Fanuc TP program (LS listing): test_parallel_centered.ls

/PROG  test_parallel_centered
/ATTR
COMMENT	= "19-02-13 13:08:30";
PROG_SIZE	= 0;
DEFAULT_GROUP	= 1, 1, *, *, *;
/APPL
    ARC Welding Equipment: 1, *, *, *, *;
/MN
   1:  CALL HOME_ALL;
   1:  UFRAME_NUM = 1;
   1:  UTOOL_NUM = 3;
   1:  COL GUARD ADJUST 150;
   1:  PR[91] = PR[90];
   1:  ! Sicherheitspunkt;
   1:  PR[92] = PR[90];
   1:  PR[92] = PR[GP1:92,3] + 50;
   1:J PR[92];
   1:  PR[GP1:91,1] = PR[GP1:90,1] + -24.070;
   1:  PR[GP1:91,2] = PR[GP1:90,2] + -16.563;
   1:  PR[GP1:91,3] = PR[GP1:90,3] + 1.100;
   1:L PR[91] 10mm/sec CNT100;
   1:  PR[GP1:91,1] = PR[GP1:90,1] + -23.760;
   1:  PR[GP1:91,2] = PR[GP1:90,2] + -16.616;
   1:L PR[91] 10mm/sec CNT100;
   1:  PR[GP1:91,1] = PR[GP1:90,1] + -18.882;
   1:  PR[GP1:91,2] = PR[GP1:90,2] + -17.045;
   1:L PR[91] 10mm/sec CNT100;
   1:  PR[GP1:91,1] = PR[GP1:90,1] + -18.568;
   1:  PR[GP1:91,2] = PR[GP1:90,2] + -17.047;
   1:L PR[91] 10mm/sec CNT100;
   1:  PR[GP1:91,1] = PR[GP1:90,1] + -18.257;
   1:  PR[GP1:91,2] = PR[GP1:90,2] + -16.997;
   1:L PR[91] 10mm/sec CNT100;
   1:  PR[GP1:91,1] = PR[GP1:90,1] + -13.503;
   1:  PR[GP1:91,2] = PR[GP1:90,2] + -15.824;
   1:L PR[91] 10mm/sec CNT100;
   1:  PR[GP1:91,1] = PR[GP1:90,1] + -13.205;
   1:  PR[GP1:91,2] = PR[GP1:90,2] + -15.724;
   1:L PR[91] 10mm/sec CNT100;
   1:  PR[GP1:91,1] = PR[GP1:90,1] + -12.928;
   1:  PR[GP1:91,2] = PR[GP1:90,2] + -15.576;
   1:L PR[91] 10mm/sec CNT100;
   1:  PR[GP1:91,1] = PR[GP1:90,1] + -8.809;
   1:  PR[GP1:91,2] = PR[GP1:90,2] + -12.928;
   1:L PR[91] 10mm/sec CNT100;
   1:  PR[GP1:91,1] = PR[GP1:90,1] + -8.559;
   1:  PR[GP1:91,2] = PR[GP1:90,2] + -12.737;
   1:L PR[91] 10mm/sec CNT100;
   1:  PR[GP1:91,1] = PR[GP1:90,1] + -8.344;
   1:  PR[GP1:91,2] = PR[GP1:90,2] + -12.508;
   1:L PR[91] 10mm/sec CNT100;
   1:  PR[GP1:91,1] = PR[GP1:90,1] + -5.304;
   1:  PR[GP1:91,2] = PR[GP1:90,2] + -8.669;
   1:L PR[91] 10mm/sec CNT100;
   1:  PR[GP1:91,1] = PR[GP1:90,1] + -5.129;
   1:  PR[GP1:91,2] = PR[GP1:90,2] + -8.408;
   1:L PR[91] 10mm/sec CNT100;
   1:  PR[GP1:91,1] = PR[GP1:90,1] + -5.000;
   1:  PR[GP1:91,2] = PR[GP1:90,2] + -8.121;
   1:L PR[91] 10mm/sec CNT100;
   1:  PR[GP1:91,1] = PR[GP1:90,1] + -3.366;
   1:  PR[GP1:91,2] = PR[GP1:90,2] + -3.509;
   1:L PR[91] 10mm/sec CNT100;
   1:  PR[GP1:91,1] = PR[GP1:90,1] + -3.259;
   1:  PR[GP1:91,2] = PR[GP1:90,2] + -3.105;
   1:L PR[91] 10mm/sec CNT100;
   1:  PR[GP1:91,1] = PR[GP1:90,1] + -2.720;
   1:  PR[GP1:91,2] = PR[GP1:90,2] + -1.858;
   1:L PR[91] 10mm/sec CNT100;
   1:  PR[GP1:91,1] = PR[GP1:90,1] + -1.598;
   1:  PR[GP1:91,2] = PR[GP1:90,2] + -0.918;
   1:L PR[91] 10mm/sec CNT100;
   1:  PR[GP1:91,1] = PR[GP1:90,1] + -0.249;
   1:  PR[GP1:91,2] = PR[GP1:90,2] + -0.599;
   1:L PR[91] 10mm/sec CNT100;
   1:  PR[GP1:91,1] = PR[GP1:90,1] + 0.522;
   1:L PR[91] 10mm/sec CNT100;
   1:  PR[GP1:91,1] = PR[GP1:90,1] + 1.871;
   1:  PR[GP1:91,2] = PR[GP1:90,2] + -0.918;
   1:L PR[91] 10mm/sec CNT100;
   1:  PR[GP1:91,1] = PR[GP1:90,1] + 2.993;
   1:  PR[GP1:91,2] = PR[GP1:90,2] + -1.858;
   1:L PR[91] 10mm/sec CNT100;
   1:  PR[GP1:91,1] = PR[GP1:90,1] + 3.521;
   1:  PR[GP1:91,2] = PR[GP1:90,2] + -3.080;
   1:L PR[91] 10mm/sec CNT100;
   1:  PR[GP1:91,1] = PR[GP1:90,1] + 5.193;
   1:  PR[GP1:91,2] = PR[GP1:90,2] + -7.798;
   1:L PR[91] 10mm/sec CNT100;
   1:  PR[GP1:91,1] = PR[GP1:90,1] + 5.253;
   1:  PR[GP1:91,2] = PR[GP1:90,2] + -8.055;
   1:L PR[91] 10mm/sec CNT100;
   1:  PR[GP1:91,1] = PR[GP1:90,1] + 5.317;
   1:  PR[GP1:91,2] = PR[GP1:90,2] + -8.236;
   1:L PR[91] 10mm/sec CNT100;
   1:  PR[GP1:91,1] = PR[GP1:90,1] + 5.385;
   1:  PR[GP1:91,2] = PR[GP1:90,2] + -8.375;
   1:L PR[91] 10mm/sec CNT100;
   1:  PR[GP1:91,1] = PR[GP1:90,1] + 8.437;
   1:  PR[GP1:91,2] = PR[GP1:90,2] + -12.228;
   1:L PR[91] 10mm/sec CNT100;
   1:  PR[GP1:91,1] = PR[GP1:90,1] + 8.577;
   1:  PR[GP1:91,2] = PR[GP1:90,2] + -12.452;
   1:L PR[91] 10mm/sec CNT100;
   1:  PR[GP1:91,1] = PR[GP1:90,1] + 8.696;
   1:  PR[GP1:91,2] = PR[GP1:90,2] + -12.602;
   1:L PR[91] 10mm/sec CNT100;
   1:  PR[GP1:91,1] = PR[GP1:90,1] + 8.805;
   1:  PR[GP1:91,2] = PR[GP1:90,2] + -12.712;
   1:L PR[91] 10mm/sec CNT100;
   1:  PR[GP1:91,1] = PR[GP1:90,1] + 12.939;
   1:  PR[GP1:91,2] = PR[GP1:90,2] + -15.370;
   1:L PR[91] 10mm/sec CNT100;
   1:  PR[GP1:91,1] = PR[GP1:90,1] + 13.144;
   1:  PR[GP1:91,2] = PR[GP1:90,2] + -15.536;
   1:L PR[91] 10mm/sec CNT100;
   1:  PR[GP1:91,1] = PR[GP1:90,1] + 13.306;
   1:  PR[GP1:91,2] = PR[GP1:90,2] + -15.640;
   1:L PR[91] 10mm/sec CNT100;
   1:  PR[GP1:91,1] = PR[GP1:90,1] + 13.444;
   1:  PR[GP1:91,2] = PR[GP1:90,2] + -15.709;
   1:L PR[91] 10mm/sec CNT100;
   1:  PR[GP1:91,1] = PR[GP1:90,1] + 18.216;
   1:  PR[GP1:91,2] = PR[GP1:90,2] + -16.885;
   1:L PR[91] 10mm/sec CNT100;
   1:  PR[GP1:91,1] = PR[GP1:90,1] + 18.464;
   1:  PR[GP1:91,2] = PR[GP1:90,2] + -16.976;
   1:L PR[91] 10mm/sec CNT100;
   1:  PR[GP1:91,1] = PR[GP1:90,1] + 18.650;
   1:  PR[GP1:91,2] = PR[GP1:90,2] + -17.022;
   1:L PR[91] 10mm/sec CNT100;
   1:  PR[GP1:91,1] = PR[GP1:90,1] + 18.803;
   1:  PR[GP1:91,2] = PR[GP1:90,2] + -17.043;
   1:L PR[91] 10mm/sec CNT100;
   1:  PR[GP1:91,1] = PR[GP1:90,1] + 23.699;
   1:  PR[GP1:91,2] = PR[GP1:90,2] + -16.613;
   1:L PR[91] 10mm/sec CNT100;
   1:  PR[GP1:91,1] = PR[GP1:90,1] + 23.963;
   1:  PR[GP1:91,2] = PR[GP1:90,2] + -16.618;
   1:L PR[91] 10mm/sec CNT100;
   1:  PR[GP1:91,1] = PR[GP1:90,1] + 24.154;
   1:  PR[GP1:91,2] = PR[GP1:90,2] + -16.602;
   1:L PR[91] 10mm/sec CNT100;
   1:  PR[GP1:91,1] = PR[GP1:90,1] + 24.306;
   1:  PR[GP1:91,2] = PR[GP1:90,2] + -16.571;
   1:L PR[91] 10mm/sec CNT100;
   1:  PR[GP1:91,1] = PR[GP1:90,1] + 28.799;
   1:  PR[GP1:91,2] = PR[GP1:90,2] + -14.580;
   1:L PR[91] 10mm/sec CNT100;
   1:  PR[GP1:91,1] = PR[GP1:90,1] + 29.051;
   1:  PR[GP1:91,2] = PR[GP1:90,2] + -14.500;
   1:L PR[91] 10mm/sec CNT100;
   1:  PR[GP1:91,1] = PR[GP1:90,1] + 29.226;
   1:  PR[GP1:91,2] = PR[GP1:90,2] + -14.422;
   1:L PR[91] 10mm/sec CNT100;
   1:  PR[GP1:91,1] = PR[GP1:90,1] + 29.360;
   1:  PR[GP1:91,2] = PR[GP1:90,2] + -14.344;
   1:L PR[91] 10mm/sec CNT100;
   1:  PR[GP1:91,1] = PR[GP1:90,1] + 32.968;
   1:  PR[GP1:91,2] = PR[GP1:90,2] + -11.006;
   1:L PR[91] 10mm/sec CNT100;
   1:  PR[GP1:91,1] = PR[GP1:90,1] + 33.180;
   1:  PR[GP1:91,2] = PR[GP1:90,2] + -10.849;
   1:L PR[91] 10mm/sec CNT100;
   1:  PR[GP1:91,1] = PR[GP1:90,1] + 33.321;
   1:  PR[GP1:91,2] = PR[GP1:90,2] + -10.719;
   1:L PR[91] 10mm/sec CNT100;
   1:  PR[GP1:91,1] = PR[GP1:90,1] + 33.422;
   1:  PR[GP1:91,2] = PR[GP1:90,2] + -10.601;
   1:L PR[91] 10mm/sec CNT100;
   1:  PR[GP1:91,1] = PR[GP1:90,1] + 35.756;
   1:  PR[GP1:91,2] = PR[GP1:90,2] + -6.274;
   1:L PR[91] 10mm/sec CNT100;
   1:  PR[GP1:91,1] = PR[GP1:90,1] + 35.906;
   1:  PR[GP1:91,2] = PR[GP1:90,2] + -6.057;
   1:L PR[91] 10mm/sec CNT100;
   1:  PR[GP1:91,1] = PR[GP1:90,1] + 35.997;
   1:  PR[GP1:91,2] = PR[GP1:90,2] + -5.888;
   1:L PR[91] 10mm/sec CNT100;
   1:  PR[GP1:91,1] = PR[GP1:90,1] + 36.055;
   1:  PR[GP1:91,2] = PR[GP1:90,2] + -5.744;
   1:L PR[91] 10mm/sec CNT100;
   1:  PR[GP1:91,1] = PR[GP1:90,1] + 36.862;
   1:  PR[GP1:91,2] = PR[GP1:90,2] + -0.893;
   1:L PR[91] 10mm/sec CNT100;
   1:  PR[GP1:91,1] = PR[GP1:90,1] + 36.933;
   1:  PR[GP1:91,2] = PR[GP1:90,2] + -0.639;
   1:L PR[91] 10mm/sec CNT100;
   1:  PR[GP1:91,1] = PR[GP1:90,1] + 36.965;
   1:  PR[GP1:91,2] = PR[GP1:90,2] + -0.450;
   1:L PR[91] 10mm/sec CNT100;
   1:  PR[GP1:91,1] = PR[GP1:90,1] + 36.973;
   1:  PR[GP1:91,2] = PR[GP1:90,2] + -0.295;
   1:L PR[91] 10mm/sec CNT100;
   1:  PR[GP1:91,1] = PR[GP1:90,1] + 36.169;
   1:  PR[GP1:91,2] = PR[GP1:90,2] + 4.541;
   1:L PR[91] 10mm/sec CNT100;
   1:  PR[GP1:91,1] = PR[GP1:90,1] + 36.125;
   1:  PR[GP1:91,2] = PR[GP1:90,2] + 4.981;
   1:L PR[91] 10mm/sec CNT100;
   1:  PR[GP1:91,1] = PR[GP1:90,1] + 36.065;
   1:  PR[GP1:91,2] = PR[GP1:90,2] + 5.203;
   1:L PR[91] 10mm/sec CNT100;
   1:  PR[GP1:91,1] = PR[GP1:90,1] + 36.036;
   1:  PR[GP1:91,2] = PR[GP1:90,2] + 5.281;
   1:L PR[91] 10mm/sec CNT100;
   1:  PR[GP1:91,1] = PR[GP1:90,1] + 33.501;
   1:  PR[GP1:91,2] = PR[GP1:90,2] + 9.982;
   1:L PR[91] 10mm/sec CNT100;
   1:  PR[GP1:91,1] = PR[GP1:90,1] + 33.453;
   1:  PR[GP1:91,2] = PR[GP1:90,2] + 10.048;
   1:L PR[91] 10mm/sec CNT100;
   1:  PR[GP1:91,1] = PR[GP1:90,1] + 33.285;
   1:  PR[GP1:91,2] = PR[GP1:90,2] + 10.237;
   1:L PR[91] 10mm/sec CNT100;
   1:  PR[GP1:91,1] = PR[GP1:90,1] + 29.691;
   1:  PR[GP1:91,2] = PR[GP1:90,2] + 13.563;
   1:L PR[91] 10mm/sec CNT100;
   1:  PR[GP1:91,1] = PR[GP1:90,1] + 29.406;
   1:  PR[GP1:91,2] = PR[GP1:90,2] + 13.794;
   1:L PR[91] 10mm/sec CNT100;
   1:  PR[GP1:91,1] = PR[GP1:90,1] + 24.940;
   1:  PR[GP1:91,2] = PR[GP1:90,2] + 15.773;
   1:L PR[91] 10mm/sec CNT100;
   1:  PR[GP1:91,1] = PR[GP1:90,1] + 24.548;
   1:  PR[GP1:91,2] = PR[GP1:90,2] + 15.978;
   1:L PR[91] 10mm/sec CNT100;
   1:  PR[GP1:91,1] = PR[GP1:90,1] + 24.331;
   1:  PR[GP1:91,2] = PR[GP1:90,2] + 16.049;
   1:L PR[91] 10mm/sec CNT100;
   1:  PR[GP1:91,1] = PR[GP1:90,1] + 24.248;
   1:  PR[GP1:91,2] = PR[GP1:90,2] + 16.068;
   1:L PR[91] 10mm/sec CNT100;
   1:  PR[GP1:91,1] = PR[GP1:90,1] + 18.930;
   1:  PR[GP1:91,2] = PR[GP1:90,2] + 16.535;
   1:L PR[91] 10mm/sec CNT100;
   1:  PR[GP1:91,1] = PR[GP1:90,1] + 18.851;
   1:  PR[GP1:91,2] = PR[GP1:90,2] + 16.531;
   1:L PR[91] 10mm/sec CNT100;
   1:  PR[GP1:91,1] = PR[GP1:90,1] + 18.598;
   1:  PR[GP1:91,2] = PR[GP1:90,2] + 16.495;
   1:L PR[91] 10mm/sec CNT100;
   1:  PR[GP1:91,1] = PR[GP1:90,1] + 13.844;
   1:  PR[GP1:91,2] = PR[GP1:90,2] + 15.322;
   1:L PR[91] 10mm/sec CNT100;
   1:  PR[GP1:91,1] = PR[GP1:90,1] + 13.499;
   1:  PR[GP1:91,2] = PR[GP1:90,2] + 15.212;
   1:L PR[91] 10mm/sec CNT100;
   1:  PR[GP1:91,1] = PR[GP1:90,1] + 9.386;
   1:  PR[GP1:91,2] = PR[GP1:90,2] + 12.569;
   1:L PR[91] 10mm/sec CNT100;
   1:  PR[GP1:91,1] = PR[GP1:90,1] + 9.000;
   1:  PR[GP1:91,2] = PR[GP1:90,2] + 12.354;
   1:L PR[91] 10mm/sec CNT100;
   1:  PR[GP1:91,1] = PR[GP1:90,1] + 8.823;
   1:  PR[GP1:91,2] = PR[GP1:90,2] + 12.214;
   1:L PR[91] 10mm/sec CNT100;
   1:  PR[GP1:91,1] = PR[GP1:90,1] + 8.760;
   1:  PR[GP1:91,2] = PR[GP1:90,2] + 12.153;
   1:L PR[91] 10mm/sec CNT100;
   1:  PR[GP1:91,1] = PR[GP1:90,1] + 5.445;
   1:  PR[GP1:91,2] = PR[GP1:90,2] + 7.967;
   1:L PR[91] 10mm/sec CNT100;
   1:  PR[GP1:91,1] = PR[GP1:90,1] + 5.406;
   1:  PR[GP1:91,2] = PR[GP1:90,2] + 7.901;
   1:L PR[91] 10mm/sec CNT100;
   1:  PR[GP1:91,1] = PR[GP1:90,1] + 5.297;
   1:  PR[GP1:91,2] = PR[GP1:90,2] + 7.667;
   1:L PR[91] 10mm/sec CNT100;
   1:  PR[GP1:91,1] = PR[GP1:90,1] + 3.662;
   1:  PR[GP1:91,2] = PR[GP1:90,2] + 3.055;
   1:L PR[91] 10mm/sec CNT100;
   1:  PR[GP1:91,1] = PR[GP1:90,1] + 3.530;
   1:  PR[GP1:91,2] = PR[GP1:90,2] + 2.582;
   1:L PR[91] 10mm/sec CNT100;
   1:  PR[GP1:91,1] = PR[GP1:90,1] + 2.993;
   1:  PR[GP1:91,2] = PR[GP1:90,2] + 1.341;
   1:L PR[91] 10mm/sec CNT100;
   1:  PR[GP1:91,1] = PR[GP1:90,1] + 1.871;
   1:  PR[GP1:91,2] = PR[GP1:90,2] + 0.401;
   1:L PR[91] 10mm/sec CNT100;
   1:  PR[GP1:91,1] = PR[GP1:90,1] + 0.522;
   1:  PR[GP1:91,2] = PR[GP1:90,2] + 0.081;
   1:L PR[91] 10mm/sec CNT100;
   1:  PR[GP1:91,1] = PR[GP1:90,1] + -0.249;
   1:L PR[91] 10mm/sec CNT100;
   1:  PR[GP1:91,1] = PR[GP1:90,1] + -1.598;
   1:  PR[GP1:91,2] = PR[GP1:90,2] + 0.401;
   1:L PR[91] 10mm/sec CNT100;
   1:  PR[GP1:91,1] = PR[GP1:90,1] + -2.720;
   1:  PR[GP1:91,2] = PR[GP1:90,2] + 1.341;
   1:L PR[91] 10mm/sec CNT100;
   1:  PR[GP1:91,1] = PR[GP1:90,1] + -3.248;
   1:  PR[GP1:91,2] = PR[GP1:90,2] + 2.562;
   1:L PR[91] 10mm/sec CNT100;
   1:  PR[GP1:91,1] = PR[GP1:90,1] + -4.917;
   1:  PR[GP1:91,2] = PR[GP1:90,2] + 7.272;
   1:L PR[91] 10mm/sec CNT100;
   1:  PR[GP1:91,1] = PR[GP1:90,1] + -5.012;
   1:  PR[GP1:91,2] = PR[GP1:90,2] + 7.629;
   1:L PR[91] 10mm/sec CNT100;
   1:  PR[GP1:91,1] = PR[GP1:90,1] + -5.118;
   1:  PR[GP1:91,2] = PR[GP1:90,2] + 7.865;
   1:L PR[91] 10mm/sec CNT100;
   1:  PR[GP1:91,1] = PR[GP1:90,1] + -8.158;
   1:  PR[GP1:91,2] = PR[GP1:90,2] + 11.704;
   1:L PR[91] 10mm/sec CNT100;
   1:  PR[GP1:91,1] = PR[GP1:90,1] + -8.363;
   1:  PR[GP1:91,2] = PR[GP1:90,2] + 12.010;
   1:L PR[91] 10mm/sec CNT100;
   1:  PR[GP1:91,1] = PR[GP1:90,1] + -8.540;
   1:  PR[GP1:91,2] = PR[GP1:90,2] + 12.200;
   1:L PR[91] 10mm/sec CNT100;
   1:  PR[GP1:91,1] = PR[GP1:90,1] + -12.659;
   1:  PR[GP1:91,2] = PR[GP1:90,2] + 14.848;
   1:L PR[91] 10mm/sec CNT100;
   1:  PR[GP1:91,1] = PR[GP1:90,1] + -12.952;
   1:  PR[GP1:91,2] = PR[GP1:90,2] + 15.072;
   1:L PR[91] 10mm/sec CNT100;
   1:  PR[GP1:91,1] = PR[GP1:90,1] + -13.181;
   1:  PR[GP1:91,2] = PR[GP1:90,2] + 15.194;
   1:L PR[91] 10mm/sec CNT100;
   1:  PR[GP1:91,1] = PR[GP1:90,1] + -17.935;
   1:  PR[GP1:91,2] = PR[GP1:90,2] + 16.366;
   1:L PR[91] 10mm/sec CNT100;
   1:  PR[GP1:91,1] = PR[GP1:90,1] + -18.284;
   1:  PR[GP1:91,2] = PR[GP1:90,2] + 16.484;
   1:L PR[91] 10mm/sec CNT100;
   1:  PR[GP1:91,1] = PR[GP1:90,1] + -18.541;
   1:  PR[GP1:91,2] = PR[GP1:90,2] + 16.525;
   1:L PR[91] 10mm/sec CNT100;
   1:  PR[GP1:91,1] = PR[GP1:90,1] + -23.418;
   1:  PR[GP1:91,2] = PR[GP1:90,2] + 16.096;
   1:L PR[91] 10mm/sec CNT100;
   1:  PR[GP1:91,1] = PR[GP1:90,1] + -23.787;
   1:  PR[GP1:91,2] = PR[GP1:90,2] + 16.094;
   1:L PR[91] 10mm/sec CNT100;
   1:  PR[GP1:91,1] = PR[GP1:90,1] + -24.043;
   1:  PR[GP1:91,2] = PR[GP1:90,2] + 16.050;
   1:L PR[91] 10mm/sec CNT100;
   1:  PR[GP1:91,1] = PR[GP1:90,1] + -28.520;
   1:  PR[GP1:91,2] = PR[GP1:90,2] + 14.065;
   1:L PR[91] 10mm/sec CNT100;
   1:  PR[GP1:91,1] = PR[GP1:90,1] + -28.868;
   1:  PR[GP1:91,2] = PR[GP1:90,2] + 13.944;
   1:L PR[91] 10mm/sec CNT100;
   1:  PR[GP1:91,1] = PR[GP1:90,1] + -29.096;
   1:  PR[GP1:91,2] = PR[GP1:90,2] + 13.820;
   1:L PR[91] 10mm/sec CNT100;
   1:  PR[GP1:91,1] = PR[GP1:90,1] + -32.690;
   1:  PR[GP1:91,2] = PR[GP1:90,2] + 10.493;
   1:L PR[91] 10mm/sec CNT100;
   1:  PR[GP1:91,1] = PR[GP1:90,1] + -32.980;
   1:  PR[GP1:91,2] = PR[GP1:90,2] + 10.266;
   1:L PR[91] 10mm/sec CNT100;
   1:  PR[GP1:91,1] = PR[GP1:90,1] + -33.155;
   1:  PR[GP1:91,2] = PR[GP1:90,2] + 10.074;
   1:L PR[91] 10mm/sec CNT100;
   1:  PR[GP1:91,1] = PR[GP1:90,1] + -35.479;
   1:  PR[GP1:91,2] = PR[GP1:90,2] + 5.763;
   1:L PR[91] 10mm/sec CNT100;
   1:  PR[GP1:91,1] = PR[GP1:90,1] + -35.680;
   1:  PR[GP1:91,2] = PR[GP1:90,2] + 5.454;
   1:L PR[91] 10mm/sec CNT100;
   1:  PR[GP1:91,1] = PR[GP1:90,1] + -35.784;
   1:  PR[GP1:91,2] = PR[GP1:90,2] + 5.216;
   1:L PR[91] 10mm/sec CNT100;
   1:  PR[GP1:91,1] = PR[GP1:90,1] + -36.588;
   1:  PR[GP1:91,2] = PR[GP1:90,2] + 0.385;
   1:L PR[91] 10mm/sec CNT100;
   1:  PR[GP1:91,1] = PR[GP1:90,1] + -36.678;
   1:  PR[GP1:91,2] = PR[GP1:90,2] + 0.027;
   1:L PR[91] 10mm/sec CNT100;
   1:  PR[GP1:91,1] = PR[GP1:90,1] + -36.699;
   1:  PR[GP1:91,2] = PR[GP1:90,2] + -0.231;
   1:L PR[91] 10mm/sec CNT100;
   1:  PR[GP1:91,1] = PR[GP1:90,1] + -35.895;
   1:  PR[GP1:91,2] = PR[GP1:90,2] + -5.063;
   1:L PR[91] 10mm/sec CNT100;
   1:  PR[GP1:91,1] = PR[GP1:90,1] + -35.865;
   1:  PR[GP1:91,2] = PR[GP1:90,2] + -5.430;
   1:L PR[91] 10mm/sec CNT100;
   1:  PR[GP1:91,1] = PR[GP1:90,1] + -35.795;
   1:  PR[GP1:91,2] = PR[GP1:90,2] + -5.709;
   1:L PR[91] 10mm/sec CNT100;
   1:  PR[GP1:91,1] = PR[GP1:90,1] + -35.669;
   1:  PR[GP1:91,2] = PR[GP1:90,2] + -5.997;
   1:L PR[91] 10mm/sec CNT100;
   1:  PR[GP1:91,1] = PR[GP1:90,1] + -33.345;
   1:  PR[GP1:91,2] = PR[GP1:90,2] + -10.308;
   1:L PR[91] 10mm/sec CNT100;
   1:  PR[GP1:91,1] = PR[GP1:90,1] + -33.174;
   1:  PR[GP1:91,2] = PR[GP1:90,2] + -10.572;
   1:L PR[91] 10mm/sec CNT100;
   1:  PR[GP1:91,1] = PR[GP1:90,1] + -32.961;
   1:  PR[GP1:91,2] = PR[GP1:90,2] + -10.803;
   1:L PR[91] 10mm/sec CNT100;
   1:  PR[GP1:91,1] = PR[GP1:90,1] + -29.367;
   1:  PR[GP1:91,2] = PR[GP1:90,2] + -14.130;
   1:L PR[91] 10mm/sec CNT100;
   1:  PR[GP1:91,1] = PR[GP1:90,1] + -29.120;
   1:  PR[GP1:91,2] = PR[GP1:90,2] + -14.324;
   1:L PR[91] 10mm/sec CNT100;
   1:  PR[GP1:91,1] = PR[GP1:90,1] + -28.844;
   1:  PR[GP1:91,2] = PR[GP1:90,2] + -14.475;
   1:L PR[91] 10mm/sec CNT100;
   1:  PR[GP1:91,1] = PR[GP1:90,1] + -24.367;
   1:  PR[GP1:91,2] = PR[GP1:90,2] + -16.459;
   1:L PR[91] 10mm/sec CNT100;
   1:  PR[GP1:91,1] = PR[GP1:90,1] + -24.070;
   1:  PR[GP1:91,2] = PR[GP1:90,2] + -16.563;
   1:L PR[91] 10mm/sec CNT100;
   1:  PR[GP1:91,1] = PR[GP1:90,1] + -22.981;
   1:  PR[GP1:91,2] = PR[GP1:90,2] + -16.750;
   1:  PR[GP1:91,3] = PR[GP1:90,3] + 2.200;
   1:L PR[91] 10mm/sec CNT100;
   1:  PR[GP1:91,1] = PR[GP1:90,1] + -19.675;
   1:  PR[GP1:91,2] = PR[GP1:90,2] + -17.040;
   1:L PR[91] 10mm/sec CNT100;
   1:  PR[GP1:91,1] = PR[GP1:90,1] + -18.569;
   1:  PR[GP1:91,2] = PR[GP1:90,2] + -17.047;
   1:L PR[91] 10mm/sec CNT100;
   1:  PR[GP1:91,1] = PR[GP1:90,1] + -17.477;
   1:  PR[GP1:91,2] = PR[GP1:90,2] + -16.871;
   1:L PR[91] 10mm/sec CNT100;
   1:  PR[GP1:91,1] = PR[GP1:90,1] + -14.255;
   1:  PR[GP1:91,2] = PR[GP1:90,2] + -16.077;
   1:L PR[91] 10mm/sec CNT100;
   1:  PR[GP1:91,1] = PR[GP1:90,1] + -13.206;
   1:  PR[GP1:91,2] = PR[GP1:90,2] + -15.724;
   1:L PR[91] 10mm/sec CNT100;
   1:  PR[GP1:91,1] = PR[GP1:90,1] + -12.229;
   1:  PR[GP1:91,2] = PR[GP1:90,2] + -15.205;
   1:L PR[91] 10mm/sec CNT100;
   1:  PR[GP1:91,1] = PR[GP1:90,1] + -9.438;
   1:  PR[GP1:91,2] = PR[GP1:90,2] + -13.411;
   1:L PR[91] 10mm/sec CNT100;
   1:  PR[GP1:91,1] = PR[GP1:90,1] + -8.560;
   1:  PR[GP1:91,2] = PR[GP1:90,2] + -12.738;
   1:L PR[91] 10mm/sec CNT100;
   1:  PR[GP1:91,1] = PR[GP1:90,1] + -7.804;
   1:  PR[GP1:91,2] = PR[GP1:90,2] + -11.931;
   1:L PR[91] 10mm/sec CNT100;
   1:  PR[GP1:91,1] = PR[GP1:90,1] + -5.743;
   1:  PR[GP1:91,2] = PR[GP1:90,2] + -9.330;
   1:L PR[91] 10mm/sec CNT100;
   1:  PR[GP1:91,1] = PR[GP1:90,1] + -5.130;
   1:  PR[GP1:91,2] = PR[GP1:90,2] + -8.409;
   1:L PR[91] 10mm/sec CNT100;
   1:  PR[GP1:91,1] = PR[GP1:90,1] + -4.676;
   1:  PR[GP1:91,2] = PR[GP1:90,2] + -7.400;
   1:L PR[91] 10mm/sec CNT100;
   1:  PR[GP1:91,1] = PR[GP1:90,1] + -3.568;
   1:  PR[GP1:91,2] = PR[GP1:90,2] + -4.275;
   1:L PR[91] 10mm/sec CNT100;
   1:  PR[GP1:91,1] = PR[GP1:90,1] + -3.259;
   1:  PR[GP1:91,2] = PR[GP1:90,2] + -3.105;
   1:L PR[91] 10mm/sec CNT100;
   1:  PR[GP1:91,1] = PR[GP1:90,1] + -2.720;
   1:  PR[GP1:91,2] = PR[GP1:90,2] + -1.858;
   1:L PR[91] 10mm/sec CNT100;
   1:  PR[GP1:91,1] = PR[GP1:90,1] + -1.598;
   1:  PR[GP1:91,2] = PR[GP1:90,2] + -0.918;
   1:L PR[91] 10mm/sec CNT100;
   1:  PR[GP1:91,1] = PR[GP1:90,1] + -0.249;
   1:  PR[GP1:91,2] = PR[GP1:90,2] + -0.599;
   1:L PR[91] 10mm/sec CNT100;
   1:  PR[GP1:91,1] = PR[GP1:90,1] + 0.522;
   1:L PR[91] 10mm/sec CNT100;
   1:  PR[GP1:91,1] = PR[GP1:90,1] + 1.871;
   1:  PR[GP1:91,2] = PR[GP1:90,2] + -0.918;
   1:L PR[91] 10mm/sec CNT100;
   1:  PR[GP1:91,1] = PR[GP1:90,1] + 2.993;
   1:  PR[GP1:91,2] = PR[GP1:90,2] + -1.858;
   1:L PR[91] 10mm/sec CNT100;
   1:  PR[GP1:91,1] = PR[GP1:90,1] + 3.521;
   1:  PR[GP1:91,2] = PR[GP1:90,2] + -3.080;
   1:L PR[91] 10mm/sec CNT100;
   1:  PR[GP1:91,1] = PR[GP1:90,1] + 4.666;
   1:  PR[GP1:91,2] = PR[GP1:90,2] + -6.311;
   1:L PR[91] 10mm/sec CNT100;
   1:  PR[GP1:91,1] = PR[GP1:90,1] + 4.847;
   1:  PR[GP1:91,2] = PR[GP1:90,2] + -7.083;
   1:L PR[91] 10mm/sec CNT100;
   1:  PR[GP1:91,1] = PR[GP1:90,1] + 5.088;
   1:  PR[GP1:91,2] = PR[GP1:90,2] + -7.761;
   1:L PR[91] 10mm/sec CNT100;
   1:  PR[GP1:91,1] = PR[GP1:90,1] + 5.386;
   1:  PR[GP1:91,2] = PR[GP1:90,2] + -8.377;
   1:L PR[91] 10mm/sec CNT100;
   1:  PR[GP1:91,1] = PR[GP1:90,1] + 7.457;
   1:  PR[GP1:91,2] = PR[GP1:90,2] + -10.992;
   1:L PR[91] 10mm/sec CNT100;
   1:  PR[GP1:91,1] = PR[GP1:90,1] + 7.878;
   1:  PR[GP1:91,2] = PR[GP1:90,2] + -11.663;
   1:L PR[91] 10mm/sec CNT100;
   1:  PR[GP1:91,1] = PR[GP1:90,1] + 8.325;
   1:  PR[GP1:91,2] = PR[GP1:90,2] + -12.227;
   1:L PR[91] 10mm/sec CNT100;
   1:  PR[GP1:91,1] = PR[GP1:90,1] + 8.806;
   1:  PR[GP1:91,2] = PR[GP1:90,2] + -12.713;
   1:L PR[91] 10mm/sec CNT100;
   1:  PR[GP1:91,1] = PR[GP1:90,1] + 11.612;
   1:  PR[GP1:91,2] = PR[GP1:90,2] + -14.517;
   1:L PR[91] 10mm/sec CNT100;
   1:  PR[GP1:91,1] = PR[GP1:90,1] + 12.228;
   1:  PR[GP1:91,2] = PR[GP1:90,2] + -15.016;
   1:L PR[91] 10mm/sec CNT100;
   1:  PR[GP1:91,1] = PR[GP1:90,1] + 12.834;
   1:  PR[GP1:91,2] = PR[GP1:90,2] + -15.405;
   1:L PR[91] 10mm/sec CNT100;
   1:  PR[GP1:91,1] = PR[GP1:90,1] + 13.446;
   1:  PR[GP1:91,2] = PR[GP1:90,2] + -15.709;
   1:L PR[91] 10mm/sec CNT100;
   1:  PR[GP1:91,1] = PR[GP1:90,1] + 16.684;
   1:  PR[GP1:91,2] = PR[GP1:90,2] + -16.508;
   1:L PR[91] 10mm/sec CNT100;
   1:  PR[GP1:91,1] = PR[GP1:90,1] + 17.428;
   1:  PR[GP1:91,2] = PR[GP1:90,2] + -16.781;
   1:L PR[91] 10mm/sec CNT100;
   1:  PR[GP1:91,1] = PR[GP1:90,1] + 18.127;
   1:  PR[GP1:91,2] = PR[GP1:90,2] + -16.953;
   1:L PR[91] 10mm/sec CNT100;
   1:  PR[GP1:91,1] = PR[GP1:90,1] + 18.805;
   1:  PR[GP1:91,2] = PR[GP1:90,2] + -17.043;
   1:L PR[91] 10mm/sec CNT100;
   1:  PR[GP1:91,1] = PR[GP1:90,1] + 22.128;
   1:  PR[GP1:91,2] = PR[GP1:90,2] + -16.751;
   1:L PR[91] 10mm/sec CNT100;
   1:  PR[GP1:91,1] = PR[GP1:90,1] + 22.920;
   1:  PR[GP1:91,2] = PR[GP1:90,2] + -16.768;
   1:L PR[91] 10mm/sec CNT100;
   1:  PR[GP1:91,1] = PR[GP1:90,1] + 23.637;
   1:  PR[GP1:91,2] = PR[GP1:90,2] + -16.705;
   1:L PR[91] 10mm/sec CNT100;
   1:  PR[GP1:91,1] = PR[GP1:90,1] + 24.308;
   1:  PR[GP1:91,2] = PR[GP1:90,2] + -16.571;
   1:L PR[91] 10mm/sec CNT100;
   1:  PR[GP1:91,1] = PR[GP1:90,1] + 27.357;
   1:  PR[GP1:91,2] = PR[GP1:90,2] + -15.219;
   1:L PR[91] 10mm/sec CNT100;
   1:  PR[GP1:91,1] = PR[GP1:90,1] + 28.113;
   1:  PR[GP1:91,2] = PR[GP1:90,2] + -14.979;
   1:L PR[91] 10mm/sec CNT100;
   1:  PR[GP1:91,1] = PR[GP1:90,1] + 28.771;
   1:  PR[GP1:91,2] = PR[GP1:90,2] + -14.687;
   1:L PR[91] 10mm/sec CNT100;
   1:  PR[GP1:91,1] = PR[GP1:90,1] + 29.361;
   1:  PR[GP1:91,2] = PR[GP1:90,2] + -14.343;
   1:L PR[91] 10mm/sec CNT100;
   1:  PR[GP1:91,1] = PR[GP1:90,1] + 31.810;
   1:  PR[GP1:91,2] = PR[GP1:90,2] + -12.077;
   1:L PR[91] 10mm/sec CNT100;
   1:  PR[GP1:91,1] = PR[GP1:90,1] + 32.447;
   1:  PR[GP1:91,2] = PR[GP1:90,2] + -11.606;
   1:L PR[91] 10mm/sec CNT100;
   1:  PR[GP1:91,1] = PR[GP1:90,1] + 32.975;
   1:  PR[GP1:91,2] = PR[GP1:90,2] + -11.117;
   1:L PR[91] 10mm/sec CNT100;
   1:  PR[GP1:91,1] = PR[GP1:90,1] + 33.423;
   1:  PR[GP1:91,2] = PR[GP1:90,2] + -10.600;
   1:L PR[91] 10mm/sec CNT100;
   1:  PR[GP1:91,1] = PR[GP1:90,1] + 35.007;
   1:  PR[GP1:91,2] = PR[GP1:90,2] + -7.663;
   1:L PR[91] 10mm/sec CNT100;
   1:  PR[GP1:91,1] = PR[GP1:90,1] + 35.457;
   1:  PR[GP1:91,2] = PR[GP1:90,2] + -7.011;
   1:L PR[91] 10mm/sec CNT100;
   1:  PR[GP1:91,1] = PR[GP1:90,1] + 35.799;
   1:  PR[GP1:91,2] = PR[GP1:90,2] + -6.377;
   1:L PR[91] 10mm/sec CNT100;
   1:  PR[GP1:91,1] = PR[GP1:90,1] + 36.055;
   1:  PR[GP1:91,2] = PR[GP1:90,2] + -5.743;
   1:L PR[91] 10mm/sec CNT100;
   1:  PR[GP1:91,1] = PR[GP1:90,1] + 36.603;
   1:  PR[GP1:91,2] = PR[GP1:90,2] + -2.451;
   1:L PR[91] 10mm/sec CNT100;
   1:  PR[GP1:91,1] = PR[GP1:90,1] + 36.818;
   1:  PR[GP1:91,2] = PR[GP1:90,2] + -1.688;
   1:L PR[91] 10mm/sec CNT100;
   1:  PR[GP1:91,1] = PR[GP1:90,1] + 36.936;
   1:  PR[GP1:91,2] = PR[GP1:90,2] + -0.978;
   1:L PR[91] 10mm/sec CNT100;
   1:  PR[GP1:91,1] = PR[GP1:90,1] + 36.973;
   1:  PR[GP1:91,2] = PR[GP1:90,2] + -0.295;
   1:L PR[91] 10mm/sec CNT100;
   1:  PR[GP1:91,1] = PR[GP1:90,1] + 36.428;
   1:  PR[GP1:91,2] = PR[GP1:90,2] + 2.983;
   1:L PR[91] 10mm/sec CNT100;
   1:  PR[GP1:91,1] = PR[GP1:90,1] + 36.290;
   1:  PR[GP1:91,2] = PR[GP1:90,2] + 4.369;
   1:L PR[91] 10mm/sec CNT100;
   1:  PR[GP1:91,1] = PR[GP1:90,1] + 36.065;
   1:  PR[GP1:91,2] = PR[GP1:90,2] + 5.202;
   1:L PR[91] 10mm/sec CNT100;
   1:  PR[GP1:91,1] = PR[GP1:90,1] + 35.923;
   1:  PR[GP1:91,2] = PR[GP1:90,2] + 5.577;
   1:L PR[91] 10mm/sec CNT100;
   1:  PR[GP1:91,1] = PR[GP1:90,1] + 33.686;
   1:  PR[GP1:91,2] = PR[GP1:90,2] + 9.725;
   1:L PR[91] 10mm/sec CNT100;
   1:  PR[GP1:91,1] = PR[GP1:90,1] + 33.454;
   1:  PR[GP1:91,2] = PR[GP1:90,2] + 10.047;
   1:L PR[91] 10mm/sec CNT100;
   1:  PR[GP1:91,1] = PR[GP1:90,1] + 32.864;
   1:  PR[GP1:91,2] = PR[GP1:90,2] + 10.712;
   1:L PR[91] 10mm/sec CNT100;
   1:  PR[GP1:91,1] = PR[GP1:90,1] + 30.428;
   1:  PR[GP1:91,2] = PR[GP1:90,2] + 12.966;
   1:L PR[91] 10mm/sec CNT100;
   1:  PR[GP1:91,1] = PR[GP1:90,1] + 29.404;
   1:  PR[GP1:91,2] = PR[GP1:90,2] + 13.795;
   1:L PR[91] 10mm/sec CNT100;
   1:  PR[GP1:91,1] = PR[GP1:90,1] + 26.381;
   1:  PR[GP1:91,2] = PR[GP1:90,2] + 15.134;
   1:L PR[91] 10mm/sec CNT100;
   1:  PR[GP1:91,1] = PR[GP1:90,1] + 25.147;
   1:  PR[GP1:91,2] = PR[GP1:90,2] + 15.781;
   1:L PR[91] 10mm/sec CNT100;
   1:  PR[GP1:91,1] = PR[GP1:90,1] + 24.333;
   1:  PR[GP1:91,2] = PR[GP1:90,2] + 16.049;
   1:L PR[91] 10mm/sec CNT100;
   1:  PR[GP1:91,1] = PR[GP1:90,1] + 23.935;
   1:  PR[GP1:91,2] = PR[GP1:90,2] + 16.138;
   1:L PR[91] 10mm/sec CNT100;
   1:  PR[GP1:91,1] = PR[GP1:90,1] + 19.241;
   1:  PR[GP1:91,2] = PR[GP1:90,2] + 16.549;
   1:L PR[91] 10mm/sec CNT100;
   1:  PR[GP1:91,1] = PR[GP1:90,1] + 18.852;
   1:  PR[GP1:91,2] = PR[GP1:90,2] + 16.531;
   1:L PR[91] 10mm/sec CNT100;
   1:  PR[GP1:91,1] = PR[GP1:90,1] + 17.964;
   1:  PR[GP1:91,2] = PR[GP1:90,2] + 16.403;
   1:L PR[91] 10mm/sec CNT100;
   1:  PR[GP1:91,1] = PR[GP1:90,1] + 14.743;
   1:  PR[GP1:91,2] = PR[GP1:90,2] + 15.608;
   1:L PR[91] 10mm/sec CNT100;
   1:  PR[GP1:91,1] = PR[GP1:90,1] + 13.500;
   1:  PR[GP1:91,2] = PR[GP1:90,2] + 15.213;
   1:L PR[91] 10mm/sec CNT100;
   1:  PR[GP1:91,1] = PR[GP1:90,1] + 10.707;
   1:  PR[GP1:91,2] = PR[GP1:90,2] + 13.420;
   1:L PR[91] 10mm/sec CNT100;
   1:  PR[GP1:91,1] = PR[GP1:90,1] + 9.490;
   1:  PR[GP1:91,2] = PR[GP1:90,2] + 12.743;
   1:L PR[91] 10mm/sec CNT100;
   1:  PR[GP1:91,1] = PR[GP1:90,1] + 8.824;
   1:  PR[GP1:91,2] = PR[GP1:90,2] + 12.215;
   1:L PR[91] 10mm/sec CNT100;
   1:  PR[GP1:91,1] = PR[GP1:90,1] + 8.526;
   1:  PR[GP1:91,2] = PR[GP1:90,2] + 11.926;
   1:L PR[91] 10mm/sec CNT100;
   1:  PR[GP1:91,1] = PR[GP1:90,1] + 5.602;
   1:  PR[GP1:91,2] = PR[GP1:90,2] + 8.230;
   1:L PR[91] 10mm/sec CNT100;
   1:  PR[GP1:91,1] = PR[GP1:90,1] + 5.407;
   1:  PR[GP1:91,2] = PR[GP1:90,2] + 7.902;
   1:L PR[91] 10mm/sec CNT100;
   1:  PR[GP1:91,1] = PR[GP1:90,1] + 5.023;
   1:  PR[GP1:91,2] = PR[GP1:90,2] + 7.083;
   1:L PR[91] 10mm/sec CNT100;
   1:  PR[GP1:91,1] = PR[GP1:90,1] + 3.916;
   1:  PR[GP1:91,2] = PR[GP1:90,2] + 3.958;
   1:L PR[91] 10mm/sec CNT100;
   1:  PR[GP1:91,1] = PR[GP1:90,1] + 3.530;
   1:  PR[GP1:91,2] = PR[GP1:90,2] + 2.582;
   1:L PR[91] 10mm/sec CNT100;
   1:  PR[GP1:91,1] = PR[GP1:90,1] + 2.993;
   1:  PR[GP1:91,2] = PR[GP1:90,2] + 1.341;
   1:L PR[91] 10mm/sec CNT100;
   1:  PR[GP1:91,1] = PR[GP1:90,1] + 1.871;
   1:  PR[GP1:91,2] = PR[GP1:90,2] + 0.401;
   1:L PR[91] 10mm/sec CNT100;
   1:  PR[GP1:91,1] = PR[GP1:90,1] + 0.522;
   1:  PR[GP1:91,2] = PR[GP1:90,2] + 0.081;
   1:L PR[91] 10mm/sec CNT100;
   1:  PR[GP1:91,1] = PR[GP1:90,1] + -0.249;
   1:L PR[91] 10mm/sec CNT100;
   1:  PR[GP1:91,1] = PR[GP1:90,1] + -1.598;
   1:  PR[GP1:91,2] = PR[GP1:90,2] + 0.401;
   1:L PR[91] 10mm/sec CNT100;
   1:  PR[GP1:91,1] = PR[GP1:90,1] + -2.720;
   1:  PR[GP1:91,2] = PR[GP1:90,2] + 1.341;
   1:L PR[91] 10mm/sec CNT100;
   1:  PR[GP1:91,1] = PR[GP1:90,1] + -3.248;
   1:  PR[GP1:91,2] = PR[GP1:90,2] + 2.562;
   1:L PR[91] 10mm/sec CNT100;
   1:  PR[GP1:91,1] = PR[GP1:90,1] + -4.390;
   1:  PR[GP1:91,2] = PR[GP1:90,2] + 5.785;
   1:L PR[91] 10mm/sec CNT100;
   1:  PR[GP1:91,1] = PR[GP1:90,1] + -4.687;
   1:  PR[GP1:91,2] = PR[GP1:90,2] + 6.908;
   1:L PR[91] 10mm/sec CNT100;
   1:  PR[GP1:91,1] = PR[GP1:90,1] + -5.119;
   1:  PR[GP1:91,2] = PR[GP1:90,2] + 7.867;
   1:L PR[91] 10mm/sec CNT100;
   1:  PR[GP1:91,1] = PR[GP1:90,1] + -7.179;
   1:  PR[GP1:91,2] = PR[GP1:90,2] + 10.467;
   1:L PR[91] 10mm/sec CNT100;
   1:  PR[GP1:91,1] = PR[GP1:90,1] + -7.822;
   1:  PR[GP1:91,2] = PR[GP1:90,2] + 11.433;
   1:L PR[91] 10mm/sec CNT100;
   1:  PR[GP1:91,1] = PR[GP1:90,1] + -8.541;
   1:  PR[GP1:91,2] = PR[GP1:90,2] + 12.201;
   1:L PR[91] 10mm/sec CNT100;
   1:  PR[GP1:91,1] = PR[GP1:90,1] + -11.332;
   1:  PR[GP1:91,2] = PR[GP1:90,2] + 13.995;
   1:L PR[91] 10mm/sec CNT100;
   1:  PR[GP1:91,1] = PR[GP1:90,1] + -12.253;
   1:  PR[GP1:91,2] = PR[GP1:90,2] + 14.700;
   1:L PR[91] 10mm/sec CNT100;
   1:  PR[GP1:91,1] = PR[GP1:90,1] + -13.182;
   1:  PR[GP1:91,2] = PR[GP1:90,2] + 15.194;
   1:L PR[91] 10mm/sec CNT100;
   1:  PR[GP1:91,1] = PR[GP1:90,1] + -16.403;
   1:  PR[GP1:91,2] = PR[GP1:90,2] + 15.989;
   1:L PR[91] 10mm/sec CNT100;
   1:  PR[GP1:91,1] = PR[GP1:90,1] + -17.503;
   1:  PR[GP1:91,2] = PR[GP1:90,2] + 16.358;
   1:L PR[91] 10mm/sec CNT100;
   1:  PR[GP1:91,1] = PR[GP1:90,1] + -18.542;
   1:  PR[GP1:91,2] = PR[GP1:90,2] + 16.525;
   1:L PR[91] 10mm/sec CNT100;
   1:  PR[GP1:91,1] = PR[GP1:90,1] + -21.847;
   1:  PR[GP1:91,2] = PR[GP1:90,2] + 16.234;
   1:L PR[91] 10mm/sec CNT100;
   1:  PR[GP1:91,1] = PR[GP1:90,1] + -23.008;
   1:  PR[GP1:91,2] = PR[GP1:90,2] + 16.228;
   1:L PR[91] 10mm/sec CNT100;
   1:  PR[GP1:91,1] = PR[GP1:90,1] + -24.044;
   1:  PR[GP1:91,2] = PR[GP1:90,2] + 16.049;
   1:L PR[91] 10mm/sec CNT100;
   1:  PR[GP1:91,1] = PR[GP1:90,1] + -27.078;
   1:  PR[GP1:91,2] = PR[GP1:90,2] + 14.705;
   1:L PR[91] 10mm/sec CNT100;
   1:  PR[GP1:91,1] = PR[GP1:90,1] + -28.174;
   1:  PR[GP1:91,2] = PR[GP1:90,2] + 14.323;
   1:L PR[91] 10mm/sec CNT100;
   1:  PR[GP1:91,1] = PR[GP1:90,1] + -29.097;
   1:  PR[GP1:91,2] = PR[GP1:90,2] + 13.819;
   1:L PR[91] 10mm/sec CNT100;
   1:  PR[GP1:91,1] = PR[GP1:90,1] + -31.532;
   1:  PR[GP1:91,2] = PR[GP1:90,2] + 11.565;
   1:L PR[91] 10mm/sec CNT100;
   1:  PR[GP1:91,1] = PR[GP1:90,1] + -32.445;
   1:  PR[GP1:91,2] = PR[GP1:90,2] + 10.849;
   1:L PR[91] 10mm/sec CNT100;
   1:  PR[GP1:91,1] = PR[GP1:90,1] + -33.156;
   1:  PR[GP1:91,2] = PR[GP1:90,2] + 10.074;
   1:L PR[91] 10mm/sec CNT100;
   1:  PR[GP1:91,1] = PR[GP1:90,1] + -34.730;
   1:  PR[GP1:91,2] = PR[GP1:90,2] + 7.153;
   1:L PR[91] 10mm/sec CNT100;
   1:  PR[GP1:91,1] = PR[GP1:90,1] + -35.363;
   1:  PR[GP1:91,2] = PR[GP1:90,2] + 6.180;
   1:L PR[91] 10mm/sec CNT100;
   1:  PR[GP1:91,1] = PR[GP1:90,1] + -35.784;
   1:  PR[GP1:91,2] = PR[GP1:90,2] + 5.216;
   1:L PR[91] 10mm/sec CNT100;
   1:  PR[GP1:91,1] = PR[GP1:90,1] + -36.329;
   1:  PR[GP1:91,2] = PR[GP1:90,2] + 1.942;
   1:L PR[91] 10mm/sec CNT100;
   1:  PR[GP1:91,1] = PR[GP1:90,1] + -36.613;
   1:  PR[GP1:91,2] = PR[GP1:90,2] + 0.817;
   1:L PR[91] 10mm/sec CNT100;
   1:  PR[GP1:91,1] = PR[GP1:90,1] + -36.699;
   1:  PR[GP1:91,2] = PR[GP1:90,2] + -0.231;
   1:L PR[91] 10mm/sec CNT100;
   1:  PR[GP1:91,1] = PR[GP1:90,1] + -36.155;
   1:  PR[GP1:91,2] = PR[GP1:90,2] + -3.505;
   1:L PR[91] 10mm/sec CNT100;
   1:  PR[GP1:91,1] = PR[GP1:90,1] + -36.059;
   1:  PR[GP1:91,2] = PR[GP1:90,2] + -4.662;
   1:L PR[91] 10mm/sec CNT100;
   1:  PR[GP1:91,1] = PR[GP1:90,1] + -35.795;
   1:  PR[GP1:91,2] = PR[GP1:90,2] + -5.708;
   1:L PR[91] 10mm/sec CNT100;
   1:  PR[GP1:91,1] = PR[GP1:90,1] + -35.352;
   1:  PR[GP1:91,2] = PR[GP1:90,2] + -6.722;
   1:L PR[91] 10mm/sec CNT100;
   1:  PR[GP1:91,1] = PR[GP1:90,1] + -33.777;
   1:  PR[GP1:91,2] = PR[GP1:90,2] + -9.644;
   1:L PR[91] 10mm/sec CNT100;
   1:  PR[GP1:91,1] = PR[GP1:90,1] + -33.174;
   1:  PR[GP1:91,2] = PR[GP1:90,2] + -10.571;
   1:L PR[91] 10mm/sec CNT100;
   1:  PR[GP1:91,1] = PR[GP1:90,1] + -32.427;
   1:  PR[GP1:91,2] = PR[GP1:90,2] + -11.387;
   1:L PR[91] 10mm/sec CNT100;
   1:  PR[GP1:91,1] = PR[GP1:90,1] + -29.991;
   1:  PR[GP1:91,2] = PR[GP1:90,2] + -13.641;
   1:L PR[91] 10mm/sec CNT100;
   1:  PR[GP1:91,1] = PR[GP1:90,1] + -29.121;
   1:  PR[GP1:91,2] = PR[GP1:90,2] + -14.324;
   1:L PR[91] 10mm/sec CNT100;
   1:  PR[GP1:91,1] = PR[GP1:90,1] + -28.150;
   1:  PR[GP1:91,2] = PR[GP1:90,2] + -14.854;
   1:L PR[91] 10mm/sec CNT100;
   1:  PR[GP1:91,1] = PR[GP1:90,1] + -25.116;
   1:  PR[GP1:91,2] = PR[GP1:90,2] + -16.198;
   1:L PR[91] 10mm/sec CNT100;
   1:  PR[GP1:91,1] = PR[GP1:90,1] + -24.071;
   1:  PR[GP1:91,2] = PR[GP1:90,2] + -16.562;
   1:L PR[91] 10mm/sec CNT100;
   1:  PR[GP1:91,1] = PR[GP1:90,1] + -22.201;
   1:  PR[GP1:91,2] = PR[GP1:90,2] + -16.884;
   1:  PR[GP1:91,3] = PR[GP1:90,3] + 3.300;
   1:L PR[91] 10mm/sec CNT100;
   1:  PR[GP1:91,1] = PR[GP1:90,1] + -20.469;
   1:  PR[GP1:91,2] = PR[GP1:90,2] + -17.036;
   1:L PR[91] 10mm/sec CNT100;
   1:  PR[GP1:91,1] = PR[GP1:90,1] + -18.570;
   1:  PR[GP1:91,2] = PR[GP1:90,2] + -17.047;
   1:L PR[91] 10mm/sec CNT100;
   1:  PR[GP1:91,1] = PR[GP1:90,1] + -16.696;
   1:  PR[GP1:91,2] = PR[GP1:90,2] + -16.746;
   1:L PR[91] 10mm/sec CNT100;
   1:  PR[GP1:91,1] = PR[GP1:90,1] + -15.007;
   1:  PR[GP1:91,2] = PR[GP1:90,2] + -16.329;
   1:L PR[91] 10mm/sec CNT100;
   1:  PR[GP1:91,1] = PR[GP1:90,1] + -13.207;
   1:  PR[GP1:91,2] = PR[GP1:90,2] + -15.725;
   1:L PR[91] 10mm/sec CNT100;
   1:  PR[GP1:91,1] = PR[GP1:90,1] + -11.531;
   1:  PR[GP1:91,2] = PR[GP1:90,2] + -14.834;
   1:L PR[91] 10mm/sec CNT100;
   1:  PR[GP1:91,1] = PR[GP1:90,1] + -10.068;
   1:  PR[GP1:91,2] = PR[GP1:90,2] + -13.893;
   1:L PR[91] 10mm/sec CNT100;
   1:  PR[GP1:91,1] = PR[GP1:90,1] + -8.561;
   1:  PR[GP1:91,2] = PR[GP1:90,2] + -12.739;
   1:L PR[91] 10mm/sec CNT100;
   1:  PR[GP1:91,1] = PR[GP1:90,1] + -7.263;
   1:  PR[GP1:91,2] = PR[GP1:90,2] + -11.353;
   1:L PR[91] 10mm/sec CNT100;
   1:  PR[GP1:91,1] = PR[GP1:90,1] + -6.183;
   1:  PR[GP1:91,2] = PR[GP1:90,2] + -9.990;
   1:L PR[91] 10mm/sec CNT100;
   1:  PR[GP1:91,1] = PR[GP1:90,1] + -5.131;
   1:  PR[GP1:91,2] = PR[GP1:90,2] + -8.410;
   1:L PR[91] 10mm/sec CNT100;
   1:  PR[GP1:91,1] = PR[GP1:90,1] + -4.351;
   1:  PR[GP1:91,2] = PR[GP1:90,2] + -6.679;
   1:L PR[91] 10mm/sec CNT100;
   1:  PR[GP1:91,1] = PR[GP1:90,1] + -3.771;
   1:  PR[GP1:91,2] = PR[GP1:90,2] + -5.041;
   1:L PR[91] 10mm/sec CNT100;
   1:  PR[GP1:91,1] = PR[GP1:90,1] + -3.259;
   1:  PR[GP1:91,2] = PR[GP1:90,2] + -3.105;
   1:L PR[91] 10mm/sec CNT100;
   1:  PR[GP1:91,1] = PR[GP1:90,1] + -2.720;
   1:  PR[GP1:91,2] = PR[GP1:90,2] + -1.858;
   1:L PR[91] 10mm/sec CNT100;
   1:  PR[GP1:91,1] = PR[GP1:90,1] + -1.598;
   1:  PR[GP1:91,2] = PR[GP1:90,2] + -0.918;
   1:L PR[91] 10mm/sec CNT100;
   1:  PR[GP1:91,1] = PR[GP1:90,1] + -0.249;
   1:  PR[GP1:91,2] = PR[GP1:90,2] + -0.599;
   1:L PR[91] 10mm/sec CNT100;
   1:  PR[GP1:91,1] = PR[GP1:90,1] + 0.522;
   1:L PR[91] 10mm/sec CNT100;
   1:  PR[GP1:91,1] = PR[GP1:90,1] + 1.870;
   1:  PR[GP1:91,2] = PR[GP1:90,2] + -0.918;
   1:L PR[91] 10mm/sec CNT100;
   1:  PR[GP1:91,1] = PR[GP1:90,1] + 2.993;
   1:  PR[GP1:91,2] = PR[GP1:90,2] + -1.858;
   1:L PR[91] 10mm/sec CNT100;
   1:  PR[GP1:91,1] = PR[GP1:90,1] + 3.521;
   1:  PR[GP1:91,2] = PR[GP1:90,2] + -3.080;
   1:L PR[91] 10mm/sec CNT100;
   1:  PR[GP1:91,1] = PR[GP1:90,1] + 4.139;
   1:  PR[GP1:91,2] = PR[GP1:90,2] + -4.824;
   1:L PR[91] 10mm/sec CNT100;
   1:  PR[GP1:91,1] = PR[GP1:90,1] + 4.441;
   1:  PR[GP1:91,2] = PR[GP1:90,2] + -6.110;
   1:L PR[91] 10mm/sec CNT100;
   1:  PR[GP1:91,1] = PR[GP1:90,1] + 4.859;
   1:  PR[GP1:91,2] = PR[GP1:90,2] + -7.287;
   1:L PR[91] 10mm/sec CNT100;
   1:  PR[GP1:91,1] = PR[GP1:90,1] + 5.386;
   1:  PR[GP1:91,2] = PR[GP1:90,2] + -8.378;
   1:L PR[91] 10mm/sec CNT100;
   1:  PR[GP1:91,1] = PR[GP1:90,1] + 6.477;
   1:  PR[GP1:91,2] = PR[GP1:90,2] + -9.755;
   1:L PR[91] 10mm/sec CNT100;
   1:  PR[GP1:91,1] = PR[GP1:90,1] + 7.179;
   1:  PR[GP1:91,2] = PR[GP1:90,2] + -10.874;
   1:L PR[91] 10mm/sec CNT100;
   1:  PR[GP1:91,1] = PR[GP1:90,1] + 7.955;
   1:  PR[GP1:91,2] = PR[GP1:90,2] + -11.852;
   1:L PR[91] 10mm/sec CNT100;
   1:  PR[GP1:91,1] = PR[GP1:90,1] + 8.807;
   1:  PR[GP1:91,2] = PR[GP1:90,2] + -12.714;
   1:L PR[91] 10mm/sec CNT100;
   1:  PR[GP1:91,1] = PR[GP1:90,1] + 10.285;
   1:  PR[GP1:91,2] = PR[GP1:90,2] + -13.664;
   1:L PR[91] 10mm/sec CNT100;
   1:  PR[GP1:91,1] = PR[GP1:90,1] + 11.312;
   1:  PR[GP1:91,2] = PR[GP1:90,2] + -14.496;
   1:L PR[91] 10mm/sec CNT100;
   1:  PR[GP1:91,1] = PR[GP1:90,1] + 12.362;
   1:  PR[GP1:91,2] = PR[GP1:90,2] + -15.170;
   1:L PR[91] 10mm/sec CNT100;
   1:  PR[GP1:91,1] = PR[GP1:90,1] + 13.447;
   1:  PR[GP1:91,2] = PR[GP1:90,2] + -15.710;
   1:L PR[91] 10mm/sec CNT100;
   1:  PR[GP1:91,1] = PR[GP1:90,1] + 15.153;
   1:  PR[GP1:91,2] = PR[GP1:90,2] + -16.131;
   1:L PR[91] 10mm/sec CNT100;
   1:  PR[GP1:91,1] = PR[GP1:90,1] + 16.393;
   1:  PR[GP1:91,2] = PR[GP1:90,2] + -16.585;
   1:L PR[91] 10mm/sec CNT100;
   1:  PR[GP1:91,1] = PR[GP1:90,1] + 17.605;
   1:  PR[GP1:91,2] = PR[GP1:90,2] + -16.884;
   1:L PR[91] 10mm/sec CNT100;
   1:  PR[GP1:91,1] = PR[GP1:90,1] + 18.806;
   1:  PR[GP1:91,2] = PR[GP1:90,2] + -17.043;
   1:L PR[91] 10mm/sec CNT100;
   1:  PR[GP1:91,1] = PR[GP1:90,1] + 20.557;
   1:  PR[GP1:91,2] = PR[GP1:90,2] + -16.889;
   1:L PR[91] 10mm/sec CNT100;
   1:  PR[GP1:91,1] = PR[GP1:90,1] + 21.877;
   1:  PR[GP1:91,2] = PR[GP1:90,2] + -16.918;
   1:L PR[91] 10mm/sec CNT100;
   1:  PR[GP1:91,1] = PR[GP1:90,1] + 23.121;
   1:  PR[GP1:91,2] = PR[GP1:90,2] + -16.809;
   1:L PR[91] 10mm/sec CNT100;
   1:  PR[GP1:91,1] = PR[GP1:90,1] + 24.309;
   1:  PR[GP1:91,2] = PR[GP1:90,2] + -16.570;
   1:L PR[91] 10mm/sec CNT100;
   1:  PR[GP1:91,1] = PR[GP1:90,1] + 25.916;
   1:  PR[GP1:91,2] = PR[GP1:90,2] + -15.858;
   1:L PR[91] 10mm/sec CNT100;
   1:  PR[GP1:91,1] = PR[GP1:90,1] + 27.175;
   1:  PR[GP1:91,2] = PR[GP1:90,2] + -15.459;
   1:L PR[91] 10mm/sec CNT100;
   1:  PR[GP1:91,1] = PR[GP1:90,1] + 28.316;
   1:  PR[GP1:91,2] = PR[GP1:90,2] + -14.952;
   1:L PR[91] 10mm/sec CNT100;
   1:  PR[GP1:91,1] = PR[GP1:90,1] + 29.363;
   1:  PR[GP1:91,2] = PR[GP1:90,2] + -14.343;
   1:L PR[91] 10mm/sec CNT100;
   1:  PR[GP1:91,1] = PR[GP1:90,1] + 30.653;
   1:  PR[GP1:91,2] = PR[GP1:90,2] + -13.149;
   1:L PR[91] 10mm/sec CNT100;
   1:  PR[GP1:91,1] = PR[GP1:90,1] + 31.715;
   1:  PR[GP1:91,2] = PR[GP1:90,2] + -12.363;
   1:L PR[91] 10mm/sec CNT100;
   1:  PR[GP1:91,1] = PR[GP1:90,1] + 32.630;
   1:  PR[GP1:91,2] = PR[GP1:90,2] + -11.515;
   1:L PR[91] 10mm/sec CNT100;
   1:  PR[GP1:91,1] = PR[GP1:90,1] + 33.424;
   1:  PR[GP1:91,2] = PR[GP1:90,2] + -10.599;
   1:L PR[91] 10mm/sec CNT100;
   1:  PR[GP1:91,1] = PR[GP1:90,1] + 34.258;
   1:  PR[GP1:91,2] = PR[GP1:90,2] + -9.052;
   1:L PR[91] 10mm/sec CNT100;
   1:  PR[GP1:91,1] = PR[GP1:90,1] + 35.009;
   1:  PR[GP1:91,2] = PR[GP1:90,2] + -7.965;
   1:L PR[91] 10mm/sec CNT100;
   1:  PR[GP1:91,1] = PR[GP1:90,1] + 35.601;
   1:  PR[GP1:91,2] = PR[GP1:90,2] + -6.866;
   1:L PR[91] 10mm/sec CNT100;
   1:  PR[GP1:91,1] = PR[GP1:90,1] + 36.055;
   1:  PR[GP1:91,2] = PR[GP1:90,2] + -5.742;
   1:L PR[91] 10mm/sec CNT100;
   1:  PR[GP1:91,1] = PR[GP1:90,1] + 36.344;
   1:  PR[GP1:91,2] = PR[GP1:90,2] + -4.008;
   1:L PR[91] 10mm/sec CNT100;
   1:  PR[GP1:91,1] = PR[GP1:90,1] + 36.702;
   1:  PR[GP1:91,2] = PR[GP1:90,2] + -2.737;
   1:L PR[91] 10mm/sec CNT100;
   1:  PR[GP1:91,1] = PR[GP1:90,1] + 36.907;
   1:  PR[GP1:91,2] = PR[GP1:90,2] + -1.505;
   1:L PR[91] 10mm/sec CNT100;
   1:  PR[GP1:91,1] = PR[GP1:90,1] + 36.973;
   1:  PR[GP1:91,2] = PR[GP1:90,2] + -0.295;
   1:L PR[91] 10mm/sec CNT100;
   1:  PR[GP1:91,1] = PR[GP1:90,1] + 36.687;
   1:  PR[GP1:91,2] = PR[GP1:90,2] + 1.425;
   1:L PR[91] 10mm/sec CNT100;
   1:  PR[GP1:91,1] = PR[GP1:90,1] + 36.456;
   1:  PR[GP1:91,2] = PR[GP1:90,2] + 3.756;
   1:L PR[91] 10mm/sec CNT100;
   1:  PR[GP1:91,1] = PR[GP1:90,1] + 36.066;
   1:  PR[GP1:91,2] = PR[GP1:90,2] + 5.202;
   1:L PR[91] 10mm/sec CNT100;
   1:  PR[GP1:91,1] = PR[GP1:90,1] + 35.811;
   1:  PR[GP1:91,2] = PR[GP1:90,2] + 5.874;
   1:L PR[91] 10mm/sec CNT100;
   1:  PR[GP1:91,1] = PR[GP1:90,1] + 33.872;
   1:  PR[GP1:91,2] = PR[GP1:90,2] + 9.469;
   1:L PR[91] 10mm/sec CNT100;
   1:  PR[GP1:91,1] = PR[GP1:90,1] + 33.455;
   1:  PR[GP1:91,2] = PR[GP1:90,2] + 10.045;
   1:L PR[91] 10mm/sec CNT100;
   1:  PR[GP1:91,1] = PR[GP1:90,1] + 32.442;
   1:  PR[GP1:91,2] = PR[GP1:90,2] + 11.188;
   1:L PR[91] 10mm/sec CNT100;
   1:  PR[GP1:91,1] = PR[GP1:90,1] + 31.166;
   1:  PR[GP1:91,2] = PR[GP1:90,2] + 12.369;
   1:L PR[91] 10mm/sec CNT100;
   1:  PR[GP1:91,1] = PR[GP1:90,1] + 29.403;
   1:  PR[GP1:91,2] = PR[GP1:90,2] + 13.796;
   1:L PR[91] 10mm/sec CNT100;
   1:  PR[GP1:91,1] = PR[GP1:90,1] + 27.823;
   1:  PR[GP1:91,2] = PR[GP1:90,2] + 14.496;
   1:L PR[91] 10mm/sec CNT100;
   1:  PR[GP1:91,1] = PR[GP1:90,1] + 25.746;
   1:  PR[GP1:91,2] = PR[GP1:90,2] + 15.584;
   1:L PR[91] 10mm/sec CNT100;
   1:  PR[GP1:91,1] = PR[GP1:90,1] + 24.335;
   1:  PR[GP1:91,2] = PR[GP1:90,2] + 16.049;
   1:L PR[91] 10mm/sec CNT100;
   1:  PR[GP1:91,1] = PR[GP1:90,1] + 23.621;
   1:  PR[GP1:91,2] = PR[GP1:90,2] + 16.208;
   1:L PR[91] 10mm/sec CNT100;
   1:  PR[GP1:91,1] = PR[GP1:90,1] + 19.553;
   1:  PR[GP1:91,2] = PR[GP1:90,2] + 16.563;
   1:L PR[91] 10mm/sec CNT100;
   1:  PR[GP1:91,1] = PR[GP1:90,1] + 18.854;
   1:  PR[GP1:91,2] = PR[GP1:90,2] + 16.532;
   1:L PR[91] 10mm/sec CNT100;
   1:  PR[GP1:91,1] = PR[GP1:90,1] + 17.331;
   1:  PR[GP1:91,2] = PR[GP1:90,2] + 16.311;
   1:L PR[91] 10mm/sec CNT100;
   1:  PR[GP1:91,1] = PR[GP1:90,1] + 15.642;
   1:  PR[GP1:91,2] = PR[GP1:90,2] + 15.895;
   1:L PR[91] 10mm/sec CNT100;
   1:  PR[GP1:91,1] = PR[GP1:90,1] + 13.501;
   1:  PR[GP1:91,2] = PR[GP1:90,2] + 15.213;
   1:L PR[91] 10mm/sec CNT100;
   1:  PR[GP1:91,1] = PR[GP1:90,1] + 12.028;
   1:  PR[GP1:91,2] = PR[GP1:90,2] + 14.270;
   1:L PR[91] 10mm/sec CNT100;
   1:  PR[GP1:91,1] = PR[GP1:90,1] + 9.979;
   1:  PR[GP1:91,2] = PR[GP1:90,2] + 13.132;
   1:L PR[91] 10mm/sec CNT100;
   1:  PR[GP1:91,1] = PR[GP1:90,1] + 8.825;
   1:  PR[GP1:91,2] = PR[GP1:90,2] + 12.216;
   1:L PR[91] 10mm/sec CNT100;
   1:  PR[GP1:91,1] = PR[GP1:90,1] + 8.292;
   1:  PR[GP1:91,2] = PR[GP1:90,2] + 11.699;
   1:L PR[91] 10mm/sec CNT100;
   1:  PR[GP1:91,1] = PR[GP1:90,1] + 5.759;
   1:  PR[GP1:91,2] = PR[GP1:90,2] + 8.494;
   1:L PR[91] 10mm/sec CNT100;
   1:  PR[GP1:91,1] = PR[GP1:90,1] + 5.407;
   1:  PR[GP1:91,2] = PR[GP1:90,2] + 7.903;
   1:L PR[91] 10mm/sec CNT100;
   1:  PR[GP1:91,1] = PR[GP1:90,1] + 4.749;
   1:  PR[GP1:91,2] = PR[GP1:90,2] + 6.499;
   1:L PR[91] 10mm/sec CNT100;
   1:  PR[GP1:91,1] = PR[GP1:90,1] + 4.169;
   1:  PR[GP1:91,2] = PR[GP1:90,2] + 4.861;
   1:L PR[91] 10mm/sec CNT100;
   1:  PR[GP1:91,1] = PR[GP1:90,1] + 3.530;
   1:  PR[GP1:91,2] = PR[GP1:90,2] + 2.582;
   1:L PR[91] 10mm/sec CNT100;
   1:  PR[GP1:91,1] = PR[GP1:90,1] + 2.993;
   1:  PR[GP1:91,2] = PR[GP1:90,2] + 1.341;
   1:L PR[91] 10mm/sec CNT100;
   1:  PR[GP1:91,1] = PR[GP1:90,1] + 1.870;
   1:  PR[GP1:91,2] = PR[GP1:90,2] + 0.401;
   1:L PR[91] 10mm/sec CNT100;
   1:  PR[GP1:91,1] = PR[GP1:90,1] + 0.522;
   1:  PR[GP1:91,2] = PR[GP1:90,2] + 0.081;
   1:L PR[91] 10mm/sec CNT100;
   1:  PR[GP1:91,1] = PR[GP1:90,1] + -0.249;
   1:L PR[91] 10mm/sec CNT100;
   1:  PR[GP1:91,1] = PR[GP1:90,1] + -1.598;
   1:  PR[GP1:91,2] = PR[GP1:90,2] + 0.401;
   1:L PR[91] 10mm/sec CNT100;
   1:  PR[GP1:91,1] = PR[GP1:90,1] + -2.720;
   1:  PR[GP1:91,2] = PR[GP1:90,2] + 1.341;
   1:L PR[91] 10mm/sec CNT100;
   1:  PR[GP1:91,1] = PR[GP1:90,1] + -3.248;
   1:  PR[GP1:91,2] = PR[GP1:90,2] + 2.562;
   1:L PR[91] 10mm/sec CNT100;
   1:  PR[GP1:91,1] = PR[GP1:90,1] + -3.864;
   1:  PR[GP1:91,2] = PR[GP1:90,2] + 4.299;
   1:L PR[91] 10mm/sec CNT100;
   1:  PR[GP1:91,1] = PR[GP1:90,1] + -4.362;
   1:  PR[GP1:91,2] = PR[GP1:90,2] + 6.186;
   1:L PR[91] 10mm/sec CNT100;
   1:  PR[GP1:91,1] = PR[GP1:90,1] + -5.119;
   1:  PR[GP1:91,2] = PR[GP1:90,2] + 7.868;
   1:L PR[91] 10mm/sec CNT100;
   1:  PR[GP1:91,1] = PR[GP1:90,1] + -6.199;
   1:  PR[GP1:91,2] = PR[GP1:90,2] + 9.231;
   1:L PR[91] 10mm/sec CNT100;
   1:  PR[GP1:91,1] = PR[GP1:90,1] + -7.282;
   1:  PR[GP1:91,2] = PR[GP1:90,2] + 10.856;
   1:L PR[91] 10mm/sec CNT100;
   1:  PR[GP1:91,1] = PR[GP1:90,1] + -8.542;
   1:  PR[GP1:91,2] = PR[GP1:90,2] + 12.201;
   1:L PR[91] 10mm/sec CNT100;
   1:  PR[GP1:91,1] = PR[GP1:90,1] + -10.005;
   1:  PR[GP1:91,2] = PR[GP1:90,2] + 13.142;
   1:L PR[91] 10mm/sec CNT100;
   1:  PR[GP1:91,1] = PR[GP1:90,1] + -11.555;
   1:  PR[GP1:91,2] = PR[GP1:90,2] + 14.329;
   1:L PR[91] 10mm/sec CNT100;
   1:  PR[GP1:91,1] = PR[GP1:90,1] + -13.183;
   1:  PR[GP1:91,2] = PR[GP1:90,2] + 15.195;
   1:L PR[91] 10mm/sec CNT100;
   1:  PR[GP1:91,1] = PR[GP1:90,1] + -14.872;
   1:  PR[GP1:91,2] = PR[GP1:90,2] + 15.611;
   1:L PR[91] 10mm/sec CNT100;
   1:  PR[GP1:91,1] = PR[GP1:90,1] + -16.723;
   1:  PR[GP1:91,2] = PR[GP1:90,2] + 16.233;
   1:L PR[91] 10mm/sec CNT100;
   1:  PR[GP1:91,1] = PR[GP1:90,1] + -18.543;
   1:  PR[GP1:91,2] = PR[GP1:90,2] + 16.525;
   1:L PR[91] 10mm/sec CNT100;
   1:  PR[GP1:91,1] = PR[GP1:90,1] + -20.276;
   1:  PR[GP1:91,2] = PR[GP1:90,2] + 16.373;
   1:L PR[91] 10mm/sec CNT100;
   1:  PR[GP1:91,1] = PR[GP1:90,1] + -22.228;
   1:  PR[GP1:91,2] = PR[GP1:90,2] + 16.362;
   1:L PR[91] 10mm/sec CNT100;
   1:  PR[GP1:91,1] = PR[GP1:90,1] + -24.045;
   1:  PR[GP1:91,2] = PR[GP1:90,2] + 16.049;
   1:L PR[91] 10mm/sec CNT100;
   1:  PR[GP1:91,1] = PR[GP1:90,1] + -25.635;
   1:  PR[GP1:91,2] = PR[GP1:90,2] + 15.344;
   1:L PR[91] 10mm/sec CNT100;
   1:  PR[GP1:91,1] = PR[GP1:90,1] + -27.479;
   1:  PR[GP1:91,2] = PR[GP1:90,2] + 14.702;
   1:L PR[91] 10mm/sec CNT100;
   1:  PR[GP1:91,1] = PR[GP1:90,1] + -29.097;
   1:  PR[GP1:91,2] = PR[GP1:90,2] + 13.819;
   1:L PR[91] 10mm/sec CNT100;
   1:  PR[GP1:91,1] = PR[GP1:90,1] + -30.374;
   1:  PR[GP1:91,2] = PR[GP1:90,2] + 12.637;
   1:L PR[91] 10mm/sec CNT100;
   1:  PR[GP1:91,1] = PR[GP1:90,1] + -31.911;
   1:  PR[GP1:91,2] = PR[GP1:90,2] + 11.433;
   1:L PR[91] 10mm/sec CNT100;
   1:  PR[GP1:91,1] = PR[GP1:90,1] + -33.156;
   1:  PR[GP1:91,2] = PR[GP1:90,2] + 10.073;
   1:L PR[91] 10mm/sec CNT100;
   1:  PR[GP1:91,1] = PR[GP1:90,1] + -33.982;
   1:  PR[GP1:91,2] = PR[GP1:90,2] + 8.542;
   1:L PR[91] 10mm/sec CNT100;
   1:  PR[GP1:91,1] = PR[GP1:90,1] + -35.046;
   1:  PR[GP1:91,2] = PR[GP1:90,2] + 6.905;
   1:L PR[91] 10mm/sec CNT100;
   1:  PR[GP1:91,1] = PR[GP1:90,1] + -35.784;
   1:  PR[GP1:91,2] = PR[GP1:90,2] + 5.215;
   1:L PR[91] 10mm/sec CNT100;
   1:  PR[GP1:91,1] = PR[GP1:90,1] + -36.070;
   1:  PR[GP1:91,2] = PR[GP1:90,2] + 3.499;
   1:L PR[91] 10mm/sec CNT100;
   1:  PR[GP1:91,1] = PR[GP1:90,1] + -36.547;
   1:  PR[GP1:91,2] = PR[GP1:90,2] + 1.606;
   1:L PR[91] 10mm/sec CNT100;
   1:  PR[GP1:91,1] = PR[GP1:90,1] + -36.699;
   1:  PR[GP1:91,2] = PR[GP1:90,2] + -0.231;
   1:L PR[91] 10mm/sec CNT100;
   1:  PR[GP1:91,1] = PR[GP1:90,1] + -36.414;
   1:  PR[GP1:91,2] = PR[GP1:90,2] + -1.947;
   1:L PR[91] 10mm/sec CNT100;
   1:  PR[GP1:91,1] = PR[GP1:90,1] + -36.253;
   1:  PR[GP1:91,2] = PR[GP1:90,2] + -3.894;
   1:L PR[91] 10mm/sec CNT100;
   1:  PR[GP1:91,1] = PR[GP1:90,1] + -35.795;
   1:  PR[GP1:91,2] = PR[GP1:90,2] + -5.708;
   1:L PR[91] 10mm/sec CNT100;
   1:  PR[GP1:91,1] = PR[GP1:90,1] + -35.035;
   1:  PR[GP1:91,2] = PR[GP1:90,2] + -7.447;
   1:L PR[91] 10mm/sec CNT100;
   1:  PR[GP1:91,1] = PR[GP1:90,1] + -34.210;
   1:  PR[GP1:91,2] = PR[GP1:90,2] + -8.979;
   1:L PR[91] 10mm/sec CNT100;
   1:  PR[GP1:91,1] = PR[GP1:90,1] + -33.175;
   1:  PR[GP1:91,2] = PR[GP1:90,2] + -10.570;
   1:L PR[91] 10mm/sec CNT100;
   1:  PR[GP1:91,1] = PR[GP1:90,1] + -31.893;
   1:  PR[GP1:91,2] = PR[GP1:90,2] + -11.970;
   1:L PR[91] 10mm/sec CNT100;
   1:  PR[GP1:91,1] = PR[GP1:90,1] + -30.616;
   1:  PR[GP1:91,2] = PR[GP1:90,2] + -13.152;
   1:L PR[91] 10mm/sec CNT100;
   1:  PR[GP1:91,1] = PR[GP1:90,1] + -29.122;
   1:  PR[GP1:91,2] = PR[GP1:90,2] + -14.323;
   1:L PR[91] 10mm/sec CNT100;
   1:  PR[GP1:91,1] = PR[GP1:90,1] + -27.456;
   1:  PR[GP1:91,2] = PR[GP1:90,2] + -15.233;
   1:L PR[91] 10mm/sec CNT100;
   1:  PR[GP1:91,1] = PR[GP1:90,1] + -25.865;
   1:  PR[GP1:91,2] = PR[GP1:90,2] + -15.938;
   1:L PR[91] 10mm/sec CNT100;
   1:  PR[GP1:91,1] = PR[GP1:90,1] + -24.072;
   1:  PR[GP1:91,2] = PR[GP1:90,2] + -16.562;
   1:L PR[91] 10mm/sec CNT100;
   1:  PR[GP1:91,1] = PR[GP1:90,1] + -21.422;
   1:  PR[GP1:91,2] = PR[GP1:90,2] + -17.018;
   1:  PR[GP1:91,3] = PR[GP1:90,3] + 4.400;
   1:L PR[91] 10mm/sec CNT100;
   1:  PR[GP1:91,1] = PR[GP1:90,1] + -21.262;
   1:  PR[GP1:91,2] = PR[GP1:90,2] + -17.032;
   1:L PR[91] 10mm/sec CNT100;
   1:  PR[GP1:91,1] = PR[GP1:90,1] + -18.571;
   1:  PR[GP1:91,2] = PR[GP1:90,2] + -17.047;
   1:L PR[91] 10mm/sec CNT100;
   1:  PR[GP1:91,1] = PR[GP1:90,1] + -15.915;
   1:  PR[GP1:91,2] = PR[GP1:90,2] + -16.620;
   1:L PR[91] 10mm/sec CNT100;
   1:  PR[GP1:91,1] = PR[GP1:90,1] + -15.759;
   1:  PR[GP1:91,2] = PR[GP1:90,2] + -16.582;
   1:L PR[91] 10mm/sec CNT100;
   1:  PR[GP1:91,1] = PR[GP1:90,1] + -13.209;
   1:  PR[GP1:91,2] = PR[GP1:90,2] + -15.725;
   1:L PR[91] 10mm/sec CNT100;
   1:  PR[GP1:91,1] = PR[GP1:90,1] + -10.833;
   1:  PR[GP1:91,2] = PR[GP1:90,2] + -14.462;
   1:L PR[91] 10mm/sec CNT100;
   1:  PR[GP1:91,1] = PR[GP1:90,1] + -10.698;
   1:  PR[GP1:91,2] = PR[GP1:90,2] + -14.375;
   1:L PR[91] 10mm/sec CNT100;
   1:  PR[GP1:91,1] = PR[GP1:90,1] + -8.562;
   1:  PR[GP1:91,2] = PR[GP1:90,2] + -12.740;
   1:L PR[91] 10mm/sec CNT100;
   1:  PR[GP1:91,1] = PR[GP1:90,1] + -6.723;
   1:  PR[GP1:91,2] = PR[GP1:90,2] + -10.776;
   1:L PR[91] 10mm/sec CNT100;
   1:  PR[GP1:91,1] = PR[GP1:90,1] + -6.623;
   1:  PR[GP1:91,2] = PR[GP1:90,2] + -10.650;
   1:L PR[91] 10mm/sec CNT100;
   1:  PR[GP1:91,1] = PR[GP1:90,1] + -5.131;
   1:  PR[GP1:91,2] = PR[GP1:90,2] + -8.411;
   1:L PR[91] 10mm/sec CNT100;
   1:  PR[GP1:91,1] = PR[GP1:90,1] + -4.027;
   1:  PR[GP1:91,2] = PR[GP1:90,2] + -5.958;
   1:L PR[91] 10mm/sec CNT100;
   1:  PR[GP1:91,1] = PR[GP1:90,1] + -3.973;
   1:  PR[GP1:91,2] = PR[GP1:90,2] + -5.806;
   1:L PR[91] 10mm/sec CNT100;
   1:  PR[GP1:91,1] = PR[GP1:90,1] + -3.259;
   1:  PR[GP1:91,2] = PR[GP1:90,2] + -3.105;
   1:L PR[91] 10mm/sec CNT100;
   1:  PR[GP1:91,1] = PR[GP1:90,1] + -2.720;
   1:  PR[GP1:91,2] = PR[GP1:90,2] + -1.858;
   1:L PR[91] 10mm/sec CNT100;
   1:  PR[GP1:91,1] = PR[GP1:90,1] + -1.597;
   1:  PR[GP1:91,2] = PR[GP1:90,2] + -0.918;
   1:L PR[91] 10mm/sec CNT100;
   1:  PR[GP1:91,1] = PR[GP1:90,1] + -0.249;
   1:  PR[GP1:91,2] = PR[GP1:90,2] + -0.599;
   1:L PR[91] 10mm/sec CNT100;
   1:  PR[GP1:91,1] = PR[GP1:90,1] + 0.522;
   1:L PR[91] 10mm/sec CNT100;
   1:  PR[GP1:91,1] = PR[GP1:90,1] + 1.870;
   1:  PR[GP1:91,2] = PR[GP1:90,2] + -0.918;
   1:L PR[91] 10mm/sec CNT100;
   1:  PR[GP1:91,1] = PR[GP1:90,1] + 2.993;
   1:  PR[GP1:91,2] = PR[GP1:90,2] + -1.858;
   1:L PR[91] 10mm/sec CNT100;
   1:  PR[GP1:91,1] = PR[GP1:90,1] + 3.521;
   1:  PR[GP1:91,2] = PR[GP1:90,2] + -3.080;
   1:L PR[91] 10mm/sec CNT100;
   1:  PR[GP1:91,1] = PR[GP1:90,1] + 3.612;
   1:  PR[GP1:91,2] = PR[GP1:90,2] + -3.338;
   1:L PR[91] 10mm/sec CNT100;
   1:  PR[GP1:91,1] = PR[GP1:90,1] + 4.035;
   1:  PR[GP1:91,2] = PR[GP1:90,2] + -5.138;
   1:L PR[91] 10mm/sec CNT100;
   1:  PR[GP1:91,1] = PR[GP1:90,1] + 4.629;
   1:  PR[GP1:91,2] = PR[GP1:90,2] + -6.812;
   1:L PR[91] 10mm/sec CNT100;
   1:  PR[GP1:91,1] = PR[GP1:90,1] + 5.387;
   1:  PR[GP1:91,2] = PR[GP1:90,2] + -8.379;
   1:L PR[91] 10mm/sec CNT100;
   1:  PR[GP1:91,1] = PR[GP1:90,1] + 5.498;
   1:  PR[GP1:91,2] = PR[GP1:90,2] + -8.519;
   1:L PR[91] 10mm/sec CNT100;
   1:  PR[GP1:91,1] = PR[GP1:90,1] + 6.481;
   1:  PR[GP1:91,2] = PR[GP1:90,2] + -10.085;
   1:L PR[91] 10mm/sec CNT100;
   1:  PR[GP1:91,1] = PR[GP1:90,1] + 7.584;
   1:  PR[GP1:91,2] = PR[GP1:90,2] + -11.478;
   1:L PR[91] 10mm/sec CNT100;
   1:  PR[GP1:91,1] = PR[GP1:90,1] + 8.808;
   1:  PR[GP1:91,2] = PR[GP1:90,2] + -12.715;
   1:L PR[91] 10mm/sec CNT100;
   1:  PR[GP1:91,1] = PR[GP1:90,1] + 8.958;
   1:  PR[GP1:91,2] = PR[GP1:90,2] + -12.811;
   1:L PR[91] 10mm/sec CNT100;
   1:  PR[GP1:91,1] = PR[GP1:90,1] + 10.395;
   1:  PR[GP1:91,2] = PR[GP1:90,2] + -13.976;
   1:L PR[91] 10mm/sec CNT100;
   1:  PR[GP1:91,1] = PR[GP1:90,1] + 11.890;
   1:  PR[GP1:91,2] = PR[GP1:90,2] + -14.936;
   1:L PR[91] 10mm/sec CNT100;
   1:  PR[GP1:91,1] = PR[GP1:90,1] + 13.448;
   1:  PR[GP1:91,2] = PR[GP1:90,2] + -15.710;
   1:L PR[91] 10mm/sec CNT100;
   1:  PR[GP1:91,1] = PR[GP1:90,1] + 13.622;
   1:  PR[GP1:91,2] = PR[GP1:90,2] + -15.753;
   1:L PR[91] 10mm/sec CNT100;
   1:  PR[GP1:91,1] = PR[GP1:90,1] + 15.358;
   1:  PR[GP1:91,2] = PR[GP1:90,2] + -16.390;
   1:L PR[91] 10mm/sec CNT100;
   1:  PR[GP1:91,1] = PR[GP1:90,1] + 17.083;
   1:  PR[GP1:91,2] = PR[GP1:90,2] + -16.815;
   1:L PR[91] 10mm/sec CNT100;
   1:  PR[GP1:91,1] = PR[GP1:90,1] + 18.808;
   1:  PR[GP1:91,2] = PR[GP1:90,2] + -17.043;
   1:L PR[91] 10mm/sec CNT100;
   1:  PR[GP1:91,1] = PR[GP1:90,1] + 18.986;
   1:  PR[GP1:91,2] = PR[GP1:90,2] + -17.028;
   1:L PR[91] 10mm/sec CNT100;
   1:  PR[GP1:91,1] = PR[GP1:90,1] + 20.835;
   1:  PR[GP1:91,2] = PR[GP1:90,2] + -17.068;
   1:L PR[91] 10mm/sec CNT100;
   1:  PR[GP1:91,1] = PR[GP1:90,1] + 22.604;
   1:  PR[GP1:91,2] = PR[GP1:90,2] + -16.912;
   1:L PR[91] 10mm/sec CNT100;
   1:  PR[GP1:91,1] = PR[GP1:90,1] + 24.311;
   1:  PR[GP1:91,2] = PR[GP1:90,2] + -16.570;
   1:L PR[91] 10mm/sec CNT100;
   1:  PR[GP1:91,1] = PR[GP1:90,1] + 24.474;
   1:  PR[GP1:91,2] = PR[GP1:90,2] + -16.498;
   1:L PR[91] 10mm/sec CNT100;
   1:  PR[GP1:91,1] = PR[GP1:90,1] + 26.237;
   1:  PR[GP1:91,2] = PR[GP1:90,2] + -15.938;
   1:L PR[91] 10mm/sec CNT100;
   1:  PR[GP1:91,1] = PR[GP1:90,1] + 27.860;
   1:  PR[GP1:91,2] = PR[GP1:90,2] + -15.217;
   1:L PR[91] 10mm/sec CNT100;
   1:  PR[GP1:91,1] = PR[GP1:90,1] + 29.364;
   1:  PR[GP1:91,2] = PR[GP1:90,2] + -14.342;
   1:L PR[91] 10mm/sec CNT100;
   1:  PR[GP1:91,1] = PR[GP1:90,1] + 29.496;
   1:  PR[GP1:91,2] = PR[GP1:90,2] + -14.220;
   1:L PR[91] 10mm/sec CNT100;
   1:  PR[GP1:91,1] = PR[GP1:90,1] + 30.982;
   1:  PR[GP1:91,2] = PR[GP1:90,2] + -13.120;
   1:L PR[91] 10mm/sec CNT100;
   1:  PR[GP1:91,1] = PR[GP1:90,1] + 32.285;
   1:  PR[GP1:91,2] = PR[GP1:90,2] + -11.913;
   1:L PR[91] 10mm/sec CNT100;
   1:  PR[GP1:91,1] = PR[GP1:90,1] + 33.425;
   1:  PR[GP1:91,2] = PR[GP1:90,2] + -10.598;
   1:L PR[91] 10mm/sec CNT100;
   1:  PR[GP1:91,1] = PR[GP1:90,1] + 33.510;
   1:  PR[GP1:91,2] = PR[GP1:90,2] + -10.441;
   1:L PR[91] 10mm/sec CNT100;
   1:  PR[GP1:91,1] = PR[GP1:90,1] + 34.560;
   1:  PR[GP1:91,2] = PR[GP1:90,2] + -8.919;
   1:L PR[91] 10mm/sec CNT100;
   1:  PR[GP1:91,1] = PR[GP1:90,1] + 35.403;
   1:  PR[GP1:91,2] = PR[GP1:90,2] + -7.355;
   1:L PR[91] 10mm/sec CNT100;
   1:  PR[GP1:91,1] = PR[GP1:90,1] + 36.056;
   1:  PR[GP1:91,2] = PR[GP1:90,2] + -5.742;
   1:L PR[91] 10mm/sec CNT100;
   1:  PR[GP1:91,1] = PR[GP1:90,1] + 36.085;
   1:  PR[GP1:91,2] = PR[GP1:90,2] + -5.565;
   1:L PR[91] 10mm/sec CNT100;
   1:  PR[GP1:91,1] = PR[GP1:90,1] + 36.586;
   1:  PR[GP1:91,2] = PR[GP1:90,2] + -3.785;
   1:L PR[91] 10mm/sec CNT100;
   1:  PR[GP1:91,1] = PR[GP1:90,1] + 36.878;
   1:  PR[GP1:91,2] = PR[GP1:90,2] + -2.033;
   1:L PR[91] 10mm/sec CNT100;
   1:  PR[GP1:91,1] = PR[GP1:90,1] + 36.973;
   1:  PR[GP1:91,2] = PR[GP1:90,2] + -0.295;
   1:L PR[91] 10mm/sec CNT100;
   1:  PR[GP1:91,1] = PR[GP1:90,1] + 36.946;
   1:  PR[GP1:91,2] = PR[GP1:90,2] + -0.133;
   1:L PR[91] 10mm/sec CNT100;
   1:  PR[GP1:91,1] = PR[GP1:90,1] + 36.621;
   1:  PR[GP1:91,2] = PR[GP1:90,2] + 3.143;
   1:L PR[91] 10mm/sec CNT100;
   1:  PR[GP1:91,1] = PR[GP1:90,1] + 36.066;
   1:  PR[GP1:91,2] = PR[GP1:90,2] + 5.201;
   1:L PR[91] 10mm/sec CNT100;
   1:  PR[GP1:91,1] = PR[GP1:90,1] + 35.698;
   1:  PR[GP1:91,2] = PR[GP1:90,2] + 6.170;
   1:L PR[91] 10mm/sec CNT100;
   1:  PR[GP1:91,1] = PR[GP1:90,1] + 34.058;
   1:  PR[GP1:91,2] = PR[GP1:90,2] + 9.212;
   1:L PR[91] 10mm/sec CNT100;
   1:  PR[GP1:91,1] = PR[GP1:90,1] + 33.456;
   1:  PR[GP1:91,2] = PR[GP1:90,2] + 10.044;
   1:L PR[91] 10mm/sec CNT100;
   1:  PR[GP1:91,1] = PR[GP1:90,1] + 32.021;
   1:  PR[GP1:91,2] = PR[GP1:90,2] + 11.663;
   1:L PR[91] 10mm/sec CNT100;
   1:  PR[GP1:91,1] = PR[GP1:90,1] + 31.903;
   1:  PR[GP1:91,2] = PR[GP1:90,2] + 11.772;
   1:L PR[91] 10mm/sec CNT100;
   1:  PR[GP1:91,1] = PR[GP1:90,1] + 29.401;
   1:  PR[GP1:91,2] = PR[GP1:90,2] + 13.797;
   1:L PR[91] 10mm/sec CNT100;
   1:  PR[GP1:91,1] = PR[GP1:90,1] + 29.264;
   1:  PR[GP1:91,2] = PR[GP1:90,2] + 13.858;
   1:L PR[91] 10mm/sec CNT100;
   1:  PR[GP1:91,1] = PR[GP1:90,1] + 26.345;
   1:  PR[GP1:91,2] = PR[GP1:90,2] + 15.387;
   1:L PR[91] 10mm/sec CNT100;
   1:  PR[GP1:91,1] = PR[GP1:90,1] + 24.336;
   1:  PR[GP1:91,2] = PR[GP1:90,2] + 16.048;
   1:L PR[91] 10mm/sec CNT100;
   1:  PR[GP1:91,1] = PR[GP1:90,1] + 23.308;
   1:  PR[GP1:91,2] = PR[GP1:90,2] + 16.277;
   1:L PR[91] 10mm/sec CNT100;
   1:  PR[GP1:91,1] = PR[GP1:90,1] + 19.865;
   1:  PR[GP1:91,2] = PR[GP1:90,2] + 16.577;
   1:L PR[91] 10mm/sec CNT100;
   1:  PR[GP1:91,1] = PR[GP1:90,1] + 18.855;
   1:  PR[GP1:91,2] = PR[GP1:90,2] + 16.532;
   1:L PR[91] 10mm/sec CNT100;
   1:  PR[GP1:91,1] = PR[GP1:90,1] + 16.698;
   1:  PR[GP1:91,2] = PR[GP1:90,2] + 16.220;
   1:L PR[91] 10mm/sec CNT100;
   1:  PR[GP1:91,1] = PR[GP1:90,1] + 16.541;
   1:  PR[GP1:91,2] = PR[GP1:90,2] + 16.181;
   1:L PR[91] 10mm/sec CNT100;
   1:  PR[GP1:91,1] = PR[GP1:90,1] + 13.497;
   1:  PR[GP1:91,2] = PR[GP1:90,2] + 15.212;
   1:L PR[91] 10mm/sec CNT100;
   1:  PR[GP1:91,1] = PR[GP1:90,1] + 13.344;
   1:  PR[GP1:91,2] = PR[GP1:90,2] + 15.118;
   1:L PR[91] 10mm/sec CNT100;
   1:  PR[GP1:91,1] = PR[GP1:90,1] + 10.469;
   1:  PR[GP1:91,2] = PR[GP1:90,2] + 13.521;
   1:L PR[91] 10mm/sec CNT100;
   1:  PR[GP1:91,1] = PR[GP1:90,1] + 8.826;
   1:  PR[GP1:91,2] = PR[GP1:90,2] + 12.217;
   1:L PR[91] 10mm/sec CNT100;
   1:  PR[GP1:91,1] = PR[GP1:90,1] + 8.058;
   1:  PR[GP1:91,2] = PR[GP1:90,2] + 11.472;
   1:L PR[91] 10mm/sec CNT100;
   1:  PR[GP1:91,1] = PR[GP1:90,1] + 5.917;
   1:  PR[GP1:91,2] = PR[GP1:90,2] + 8.758;
   1:L PR[91] 10mm/sec CNT100;
   1:  PR[GP1:91,1] = PR[GP1:90,1] + 5.408;
   1:  PR[GP1:91,2] = PR[GP1:90,2] + 7.905;
   1:L PR[91] 10mm/sec CNT100;
   1:  PR[GP1:91,1] = PR[GP1:90,1] + 4.476;
   1:  PR[GP1:91,2] = PR[GP1:90,2] + 5.915;
   1:L PR[91] 10mm/sec CNT100;
   1:  PR[GP1:91,1] = PR[GP1:90,1] + 4.422;
   1:  PR[GP1:91,2] = PR[GP1:90,2] + 5.764;
   1:L PR[91] 10mm/sec CNT100;
   1:  PR[GP1:91,1] = PR[GP1:90,1] + 3.530;
   1:  PR[GP1:91,2] = PR[GP1:90,2] + 2.582;
   1:L PR[91] 10mm/sec CNT100;
   1:  PR[GP1:91,1] = PR[GP1:90,1] + 2.993;
   1:  PR[GP1:91,2] = PR[GP1:90,2] + 1.341;
   1:L PR[91] 10mm/sec CNT100;
   1:  PR[GP1:91,1] = PR[GP1:90,1] + 1.870;
   1:  PR[GP1:91,2] = PR[GP1:90,2] + 0.400;
   1:L PR[91] 10mm/sec CNT100;
   1:  PR[GP1:91,1] = PR[GP1:90,1] + 0.522;
   1:  PR[GP1:91,2] = PR[GP1:90,2] + 0.081;
   1:L PR[91] 10mm/sec CNT100;
   1:  PR[GP1:91,1] = PR[GP1:90,1] + -0.249;
   1:L PR[91] 10mm/sec CNT100;
   1:  PR[GP1:91,1] = PR[GP1:90,1] + -1.597;
   1:  PR[GP1:91,2] = PR[GP1:90,2] + 0.400;
   1:L PR[91] 10mm/sec CNT100;
   1:  PR[GP1:91,1] = PR[GP1:90,1] + -2.720;
   1:  PR[GP1:91,2] = PR[GP1:90,2] + 1.341;
   1:L PR[91] 10mm/sec CNT100;
   1:  PR[GP1:91,1] = PR[GP1:90,1] + -3.248;
   1:  PR[GP1:91,2] = PR[GP1:90,2] + 2.562;
   1:L PR[91] 10mm/sec CNT100;
   1:  PR[GP1:91,1] = PR[GP1:90,1] + -3.337;
   1:  PR[GP1:91,2] = PR[GP1:90,2] + 2.812;
   1:L PR[91] 10mm/sec CNT100;
   1:  PR[GP1:91,1] = PR[GP1:90,1] + -4.038;
   1:  PR[GP1:91,2] = PR[GP1:90,2] + 5.465;
   1:L PR[91] 10mm/sec CNT100;
   1:  PR[GP1:91,1] = PR[GP1:90,1] + -5.120;
   1:  PR[GP1:91,2] = PR[GP1:90,2] + 7.869;
   1:L PR[91] 10mm/sec CNT100;
   1:  PR[GP1:91,1] = PR[GP1:90,1] + -5.219;
   1:  PR[GP1:91,2] = PR[GP1:90,2] + 7.994;
   1:L PR[91] 10mm/sec CNT100;
   1:  PR[GP1:91,1] = PR[GP1:90,1] + -6.741;
   1:  PR[GP1:91,2] = PR[GP1:90,2] + 10.278;
   1:L PR[91] 10mm/sec CNT100;
   1:  PR[GP1:91,1] = PR[GP1:90,1] + -8.543;
   1:  PR[GP1:91,2] = PR[GP1:90,2] + 12.202;
   1:L PR[91] 10mm/sec CNT100;
   1:  PR[GP1:91,1] = PR[GP1:90,1] + -8.678;
   1:  PR[GP1:91,2] = PR[GP1:90,2] + 12.289;
   1:L PR[91] 10mm/sec CNT100;
   1:  PR[GP1:91,1] = PR[GP1:90,1] + -10.857;
   1:  PR[GP1:91,2] = PR[GP1:90,2] + 13.958;
   1:L PR[91] 10mm/sec CNT100;
   1:  PR[GP1:91,1] = PR[GP1:90,1] + -13.184;
   1:  PR[GP1:91,2] = PR[GP1:90,2] + 15.195;
   1:L PR[91] 10mm/sec CNT100;
   1:  PR[GP1:91,1] = PR[GP1:90,1] + -13.340;
   1:  PR[GP1:91,2] = PR[GP1:90,2] + 15.234;
   1:L PR[91] 10mm/sec CNT100;
   1:  PR[GP1:91,1] = PR[GP1:90,1] + -15.942;
   1:  PR[GP1:91,2] = PR[GP1:90,2] + 16.107;
   1:L PR[91] 10mm/sec CNT100;
   1:  PR[GP1:91,1] = PR[GP1:90,1] + -18.544;
   1:  PR[GP1:91,2] = PR[GP1:90,2] + 16.525;
   1:L PR[91] 10mm/sec CNT100;
   1:  PR[GP1:91,1] = PR[GP1:90,1] + -18.704;
   1:  PR[GP1:91,2] = PR[GP1:90,2] + 16.511;
   1:L PR[91] 10mm/sec CNT100;
   1:  PR[GP1:91,1] = PR[GP1:90,1] + -21.449;
   1:  PR[GP1:91,2] = PR[GP1:90,2] + 16.496;
   1:L PR[91] 10mm/sec CNT100;
   1:  PR[GP1:91,1] = PR[GP1:90,1] + -24.046;
   1:  PR[GP1:91,2] = PR[GP1:90,2] + 16.049;
   1:L PR[91] 10mm/sec CNT100;
   1:  PR[GP1:91,1] = PR[GP1:90,1] + -24.193;
   1:  PR[GP1:91,2] = PR[GP1:90,2] + 15.984;
   1:L PR[91] 10mm/sec CNT100;
   1:  PR[GP1:91,1] = PR[GP1:90,1] + -26.785;
   1:  PR[GP1:91,2] = PR[GP1:90,2] + 15.081;
   1:L PR[91] 10mm/sec CNT100;
   1:  PR[GP1:91,1] = PR[GP1:90,1] + -29.098;
   1:  PR[GP1:91,2] = PR[GP1:90,2] + 13.818;
   1:L PR[91] 10mm/sec CNT100;
   1:  PR[GP1:91,1] = PR[GP1:90,1] + -29.216;
   1:  PR[GP1:91,2] = PR[GP1:90,2] + 13.709;
   1:L PR[91] 10mm/sec CNT100;
   1:  PR[GP1:91,1] = PR[GP1:90,1] + -31.377;
   1:  PR[GP1:91,2] = PR[GP1:90,2] + 12.016;
   1:L PR[91] 10mm/sec CNT100;
   1:  PR[GP1:91,1] = PR[GP1:90,1] + -33.157;
   1:  PR[GP1:91,2] = PR[GP1:90,2] + 10.072;
   1:L PR[91] 10mm/sec CNT100;
   1:  PR[GP1:91,1] = PR[GP1:90,1] + -33.233;
   1:  PR[GP1:91,2] = PR[GP1:90,2] + 9.931;
   1:L PR[91] 10mm/sec CNT100;
   1:  PR[GP1:91,1] = PR[GP1:90,1] + -34.729;
   1:  PR[GP1:91,2] = PR[GP1:90,2] + 7.630;
   1:L PR[91] 10mm/sec CNT100;
   1:  PR[GP1:91,1] = PR[GP1:90,1] + -35.784;
   1:  PR[GP1:91,2] = PR[GP1:90,2] + 5.215;
   1:L PR[91] 10mm/sec CNT100;
   1:  PR[GP1:91,1] = PR[GP1:90,1] + -35.811;
   1:  PR[GP1:91,2] = PR[GP1:90,2] + 5.057;
   1:L PR[91] 10mm/sec CNT100;
   1:  PR[GP1:91,1] = PR[GP1:90,1] + -36.482;
   1:  PR[GP1:91,2] = PR[GP1:90,2] + 2.395;
   1:L PR[91] 10mm/sec CNT100;
   1:  PR[GP1:91,1] = PR[GP1:90,1] + -36.699;
   1:  PR[GP1:91,2] = PR[GP1:90,2] + -0.231;
   1:L PR[91] 10mm/sec CNT100;
   1:  PR[GP1:91,1] = PR[GP1:90,1] + -36.673;
   1:  PR[GP1:91,2] = PR[GP1:90,2] + -0.390;
   1:L PR[91] 10mm/sec CNT100;
   1:  PR[GP1:91,1] = PR[GP1:90,1] + -36.447;
   1:  PR[GP1:91,2] = PR[GP1:90,2] + -3.125;
   1:L PR[91] 10mm/sec CNT100;
   1:  PR[GP1:91,1] = PR[GP1:90,1] + -35.795;
   1:  PR[GP1:91,2] = PR[GP1:90,2] + -5.707;
   1:L PR[91] 10mm/sec CNT100;
   1:  PR[GP1:91,1] = PR[GP1:90,1] + -34.718;
   1:  PR[GP1:91,2] = PR[GP1:90,2] + -8.173;
   1:L PR[91] 10mm/sec CNT100;
   1:  PR[GP1:91,1] = PR[GP1:90,1] + -34.642;
   1:  PR[GP1:91,2] = PR[GP1:90,2] + -8.314;
   1:L PR[91] 10mm/sec CNT100;
   1:  PR[GP1:91,1] = PR[GP1:90,1] + -33.175;
   1:  PR[GP1:91,2] = PR[GP1:90,2] + -10.570;
   1:L PR[91] 10mm/sec CNT100;
   1:  PR[GP1:91,1] = PR[GP1:90,1] + -31.358;
   1:  PR[GP1:91,2] = PR[GP1:90,2] + -12.554;
   1:L PR[91] 10mm/sec CNT100;
   1:  PR[GP1:91,1] = PR[GP1:90,1] + -31.240;
   1:  PR[GP1:91,2] = PR[GP1:90,2] + -12.663;
   1:L PR[91] 10mm/sec CNT100;
   1:  PR[GP1:91,1] = PR[GP1:90,1] + -29.122;
   1:  PR[GP1:91,2] = PR[GP1:90,2] + -14.322;
   1:L PR[91] 10mm/sec CNT100;
   1:  PR[GP1:91,1] = PR[GP1:90,1] + -26.761;
   1:  PR[GP1:91,2] = PR[GP1:90,2] + -15.612;
   1:L PR[91] 10mm/sec CNT100;
   1:  PR[GP1:91,1] = PR[GP1:90,1] + -26.614;
   1:  PR[GP1:91,2] = PR[GP1:90,2] + -15.677;
   1:L PR[91] 10mm/sec CNT100;
   1:  PR[GP1:91,1] = PR[GP1:90,1] + -24.073;
   1:  PR[GP1:91,2] = PR[GP1:90,2] + -16.562;
   1:L PR[91] 10mm/sec CNT100;
   1:  PR[GP1:91,1] = PR[GP1:90,1] + -21.884;
   1:  PR[GP1:91,2] = PR[GP1:90,2] + -16.932;
   1:  PR[GP1:91,3] = PR[GP1:90,3] + 5.500;
   1:L PR[91] 10mm/sec CNT100;
   1:  PR[GP1:91,1] = PR[GP1:90,1] + -21.274;
   1:  PR[GP1:91,2] = PR[GP1:90,2] + -17.051;
   1:L PR[91] 10mm/sec CNT100;
   1:  PR[GP1:91,1] = PR[GP1:90,1] + -19.039;
   1:  PR[GP1:91,2] = PR[GP1:90,2] + -17.063;
   1:L PR[91] 10mm/sec CNT100;
   1:  PR[GP1:91,1] = PR[GP1:90,1] + -18.338;
   1:  PR[GP1:91,2] = PR[GP1:90,2] + -17.048;
   1:L PR[91] 10mm/sec CNT100;
   1:  PR[GP1:91,1] = PR[GP1:90,1] + -16.187;
   1:  PR[GP1:91,2] = PR[GP1:90,2] + -16.703;
   1:L PR[91] 10mm/sec CNT100;
   1:  PR[GP1:91,1] = PR[GP1:90,1] + -15.415;
   1:  PR[GP1:91,2] = PR[GP1:90,2] + -16.519;
   1:L PR[91] 10mm/sec CNT100;
   1:  PR[GP1:91,1] = PR[GP1:90,1] + -13.407;
   1:  PR[GP1:91,2] = PR[GP1:90,2] + -15.845;
   1:L PR[91] 10mm/sec CNT100;
   1:  PR[GP1:91,1] = PR[GP1:90,1] + -12.602;
   1:  PR[GP1:91,2] = PR[GP1:90,2] + -15.461;
   1:L PR[91] 10mm/sec CNT100;
   1:  PR[GP1:91,1] = PR[GP1:90,1] + -10.788;
   1:  PR[GP1:91,2] = PR[GP1:90,2] + -14.496;
   1:L PR[91] 10mm/sec CNT100;
   1:  PR[GP1:91,1] = PR[GP1:90,1] + -8.410;
   1:  PR[GP1:91,2] = PR[GP1:90,2] + -12.672;
   1:L PR[91] 10mm/sec CNT100;
   1:  PR[GP1:91,1] = PR[GP1:90,1] + -7.047;
   1:  PR[GP1:91,2] = PR[GP1:90,2] + -11.216;
   1:L PR[91] 10mm/sec CNT100;
   1:  PR[GP1:91,1] = PR[GP1:90,1] + -6.393;
   1:  PR[GP1:91,2] = PR[GP1:90,2] + -10.442;
   1:L PR[91] 10mm/sec CNT100;
   1:  PR[GP1:91,1] = PR[GP1:90,1] + -5.311;
   1:  PR[GP1:91,2] = PR[GP1:90,2] + -8.818;
   1:L PR[91] 10mm/sec CNT100;
   1:  PR[GP1:91,1] = PR[GP1:90,1] + -4.808;
   1:  PR[GP1:91,2] = PR[GP1:90,2] + -7.876;
   1:L PR[91] 10mm/sec CNT100;
   1:  PR[GP1:91,1] = PR[GP1:90,1] + -4.019;
   1:  PR[GP1:91,2] = PR[GP1:90,2] + -6.124;
   1:L PR[91] 10mm/sec CNT100;
   1:  PR[GP1:91,1] = PR[GP1:90,1] + -3.198;
   1:  PR[GP1:91,2] = PR[GP1:90,2] + -3.035;
   1:L PR[91] 10mm/sec CNT100;
   1:  PR[GP1:91,1] = PR[GP1:90,1] + -3.114;
   1:  PR[GP1:91,2] = PR[GP1:90,2] + -2.920;
   1:L PR[91] 10mm/sec CNT100;
   1:  PR[GP1:91,1] = PR[GP1:90,1] + -2.699;
   1:  PR[GP1:91,2] = PR[GP1:90,2] + -1.963;
   1:L PR[91] 10mm/sec CNT100;
   1:  PR[GP1:91,1] = PR[GP1:90,1] + -2.543;
   1:  PR[GP1:91,2] = PR[GP1:90,2] + -1.754;
   1:L PR[91] 10mm/sec CNT100;
   1:  PR[GP1:91,1] = PR[GP1:90,1] + -1.778;
   1:  PR[GP1:91,2] = PR[GP1:90,2] + -1.100;
   1:L PR[91] 10mm/sec CNT100;
   1:  PR[GP1:91,1] = PR[GP1:90,1] + -1.497;
   1:  PR[GP1:91,2] = PR[GP1:90,2] + -0.906;
   1:L PR[91] 10mm/sec CNT100;
   1:  PR[GP1:91,1] = PR[GP1:90,1] + -0.723;
   1:  PR[GP1:91,2] = PR[GP1:90,2] + -0.723;
   1:L PR[91] 10mm/sec CNT100;
   1:  PR[GP1:91,1] = PR[GP1:90,1] + -0.659;
   1:  PR[GP1:91,2] = PR[GP1:90,2] + -0.689;
   1:L PR[91] 10mm/sec CNT100;
   1:  PR[GP1:91,1] = PR[GP1:90,1] + -0.403;
   1:  PR[GP1:91,2] = PR[GP1:90,2] + -0.616;
   1:L PR[91] 10mm/sec CNT100;
   1:  PR[GP1:91,1] = PR[GP1:90,1] + 0.302;
   1:  PR[GP1:91,2] = PR[GP1:90,2] + -0.597;
   1:L PR[91] 10mm/sec CNT100;
   1:  PR[GP1:91,1] = PR[GP1:90,1] + 1.677;
   1:  PR[GP1:91,2] = PR[GP1:90,2] + -0.920;
   1:L PR[91] 10mm/sec CNT100;
   1:  PR[GP1:91,1] = PR[GP1:90,1] + 2.807;
   1:  PR[GP1:91,2] = PR[GP1:90,2] + -1.866;
   1:L PR[91] 10mm/sec CNT100;
   1:  PR[GP1:91,1] = PR[GP1:90,1] + 3.045;
   1:  PR[GP1:91,2] = PR[GP1:90,2] + -2.416;
   1:L PR[91] 10mm/sec CNT100;
   1:  PR[GP1:91,1] = PR[GP1:90,1] + 3.252;
   1:  PR[GP1:91,2] = PR[GP1:90,2] + -2.762;
   1:L PR[91] 10mm/sec CNT100;
   1:  PR[GP1:91,1] = PR[GP1:90,1] + 3.411;
   1:  PR[GP1:91,2] = PR[GP1:90,2] + -3.110;
   1:L PR[91] 10mm/sec CNT100;
   1:  PR[GP1:91,1] = PR[GP1:90,1] + 4.098;
   1:  PR[GP1:91,2] = PR[GP1:90,2] + -5.754;
   1:L PR[91] 10mm/sec CNT100;
   1:  PR[GP1:91,1] = PR[GP1:90,1] + 5.159;
   1:  PR[GP1:91,2] = PR[GP1:90,2] + -8.163;
   1:L PR[91] 10mm/sec CNT100;
   1:  PR[GP1:91,1] = PR[GP1:90,1] + 6.591;
   1:  PR[GP1:91,2] = PR[GP1:90,2] + -10.380;
   1:L PR[91] 10mm/sec CNT100;
   1:  PR[GP1:91,1] = PR[GP1:90,1] + 8.236;
   1:  PR[GP1:91,2] = PR[GP1:90,2] + -12.250;
   1:L PR[91] 10mm/sec CNT100;
   1:  PR[GP1:91,1] = PR[GP1:90,1] + 8.382;
   1:  PR[GP1:91,2] = PR[GP1:90,2] + -12.397;
   1:L PR[91] 10mm/sec CNT100;
   1:  PR[GP1:91,1] = PR[GP1:90,1] + 10.323;
   1:  PR[GP1:91,2] = PR[GP1:90,2] + -14.005;
   1:L PR[91] 10mm/sec CNT100;
   1:  PR[GP1:91,1] = PR[GP1:90,1] + 10.743;
   1:  PR[GP1:91,2] = PR[GP1:90,2] + -14.275;
   1:L PR[91] 10mm/sec CNT100;
   1:  PR[GP1:91,1] = PR[GP1:90,1] + 12.281;
   1:  PR[GP1:91,2] = PR[GP1:90,2] + -15.195;
   1:L PR[91] 10mm/sec CNT100;
   1:  PR[GP1:91,1] = PR[GP1:90,1] + 12.935;
   1:  PR[GP1:91,2] = PR[GP1:90,2] + -15.521;
   1:L PR[91] 10mm/sec CNT100;
   1:  PR[GP1:91,1] = PR[GP1:90,1] + 14.245;
   1:  PR[GP1:91,2] = PR[GP1:90,2] + -16.048;
   1:L PR[91] 10mm/sec CNT100;
   1:  PR[GP1:91,1] = PR[GP1:90,1] + 15.106;
   1:  PR[GP1:91,2] = PR[GP1:90,2] + -16.364;
   1:L PR[91] 10mm/sec CNT100;
   1:  PR[GP1:91,1] = PR[GP1:90,1] + 16.001;
   1:  PR[GP1:91,2] = PR[GP1:90,2] + -16.584;
   1:L PR[91] 10mm/sec CNT100;
   1:  PR[GP1:91,1] = PR[GP1:90,1] + 17.243;
   1:  PR[GP1:91,2] = PR[GP1:90,2] + -16.870;
   1:L PR[91] 10mm/sec CNT100;
   1:  PR[GP1:91,1] = PR[GP1:90,1] + 18.286;
   1:  PR[GP1:91,2] = PR[GP1:90,2] + -17.008;
   1:L PR[91] 10mm/sec CNT100;
   1:  PR[GP1:91,1] = PR[GP1:90,1] + 19.324;
   1:  PR[GP1:91,2] = PR[GP1:90,2] + -17.081;
   1:L PR[91] 10mm/sec CNT100;
   1:  PR[GP1:91,1] = PR[GP1:90,1] + 20.484;
   1:  PR[GP1:91,2] = PR[GP1:90,2] + -17.106;
   1:L PR[91] 10mm/sec CNT100;
   1:  PR[GP1:91,1] = PR[GP1:90,1] + 22.606;
   1:  PR[GP1:91,2] = PR[GP1:90,2] + -16.920;
   1:L PR[91] 10mm/sec CNT100;
   1:  PR[GP1:91,1] = PR[GP1:90,1] + 23.828;
   1:  PR[GP1:91,2] = PR[GP1:90,2] + -16.675;
   1:L PR[91] 10mm/sec CNT100;
   1:  PR[GP1:91,1] = PR[GP1:90,1] + 24.613;
   1:  PR[GP1:91,2] = PR[GP1:90,2] + -16.480;
   1:L PR[91] 10mm/sec CNT100;
   1:  PR[GP1:91,1] = PR[GP1:90,1] + 25.860;
   1:  PR[GP1:91,2] = PR[GP1:90,2] + -16.084;
   1:L PR[91] 10mm/sec CNT100;
   1:  PR[GP1:91,1] = PR[GP1:90,1] + 27.767;
   1:  PR[GP1:91,2] = PR[GP1:90,2] + -15.252;
   1:L PR[91] 10mm/sec CNT100;
   1:  PR[GP1:91,1] = PR[GP1:90,1] + 28.951;
   1:  PR[GP1:91,2] = PR[GP1:90,2] + -14.563;
   1:L PR[91] 10mm/sec CNT100;
   1:  PR[GP1:91,1] = PR[GP1:90,1] + 29.512;
   1:  PR[GP1:91,2] = PR[GP1:90,2] + -14.214;
   1:L PR[91] 10mm/sec CNT100;
   1:  PR[GP1:91,1] = PR[GP1:90,1] + 30.643;
   1:  PR[GP1:91,2] = PR[GP1:90,2] + -13.377;
   1:L PR[91] 10mm/sec CNT100;
   1:  PR[GP1:91,1] = PR[GP1:90,1] + 31.092;
   1:  PR[GP1:91,2] = PR[GP1:90,2] + -12.990;
   1:L PR[91] 10mm/sec CNT100;
   1:  PR[GP1:91,1] = PR[GP1:90,1] + 32.150;
   1:  PR[GP1:91,2] = PR[GP1:90,2] + -12.010;
   1:L PR[91] 10mm/sec CNT100;
   1:  PR[GP1:91,1] = PR[GP1:90,1] + 33.469;
   1:  PR[GP1:91,2] = PR[GP1:90,2] + -10.477;
   1:L PR[91] 10mm/sec CNT100;
   1:  PR[GP1:91,1] = PR[GP1:90,1] + 34.300;
   1:  PR[GP1:91,2] = PR[GP1:90,2] + -9.274;
   1:L PR[91] 10mm/sec CNT100;
   1:  PR[GP1:91,1] = PR[GP1:90,1] + 34.572;
   1:  PR[GP1:91,2] = PR[GP1:90,2] + -8.825;
   1:L PR[91] 10mm/sec CNT100;
   1:  PR[GP1:91,1] = PR[GP1:90,1] + 35.276;
   1:  PR[GP1:91,2] = PR[GP1:90,2] + -7.520;
   1:L PR[91] 10mm/sec CNT100;
   1:  PR[GP1:91,1] = PR[GP1:90,1] + 36.031;
   1:  PR[GP1:91,2] = PR[GP1:90,2] + -5.659;
   1:L PR[91] 10mm/sec CNT100;
   1:  PR[GP1:91,1] = PR[GP1:90,1] + 36.438;
   1:  PR[GP1:91,2] = PR[GP1:90,2] + -4.215;
   1:L PR[91] 10mm/sec CNT100;
   1:  PR[GP1:91,1] = PR[GP1:90,1] + 36.551;
   1:  PR[GP1:91,2] = PR[GP1:90,2] + -3.742;
   1:L PR[91] 10mm/sec CNT100;
   1:  PR[GP1:91,1] = PR[GP1:90,1] + 36.797;
   1:  PR[GP1:91,2] = PR[GP1:90,2] + -2.262;
   1:L PR[91] 10mm/sec CNT100;
   1:  PR[GP1:91,1] = PR[GP1:90,1] + 36.881;
   1:  PR[GP1:91,2] = PR[GP1:90,2] + -0.726;
   1:L PR[91] 10mm/sec CNT100;
   1:  PR[GP1:91,1] = PR[GP1:90,1] + 36.926;
   1:  PR[GP1:91,2] = PR[GP1:90,2] + -0.265;
   1:L PR[91] 10mm/sec CNT100;
   1:  PR[GP1:91,1] = PR[GP1:90,1] + 36.591;
   1:  PR[GP1:91,2] = PR[GP1:90,2] + 3.043;
   1:L PR[91] 10mm/sec CNT100;
   1:  PR[GP1:91,1] = PR[GP1:90,1] + 36.404;
   1:  PR[GP1:91,2] = PR[GP1:90,2] + 3.652;
   1:L PR[91] 10mm/sec CNT100;
   1:  PR[GP1:91,1] = PR[GP1:90,1] + 35.929;
   1:  PR[GP1:91,2] = PR[GP1:90,2] + 5.412;
   1:L PR[91] 10mm/sec CNT100;
   1:  PR[GP1:91,1] = PR[GP1:90,1] + 35.628;
   1:  PR[GP1:91,2] = PR[GP1:90,2] + 6.206;
   1:L PR[91] 10mm/sec CNT100;
   1:  PR[GP1:91,1] = PR[GP1:90,1] + 34.037;
   1:  PR[GP1:91,2] = PR[GP1:90,2] + 9.153;
   1:L PR[91] 10mm/sec CNT100;
   1:  PR[GP1:91,1] = PR[GP1:90,1] + 33.586;
   1:  PR[GP1:91,2] = PR[GP1:90,2] + 9.698;
   1:L PR[91] 10mm/sec CNT100;
   1:  PR[GP1:91,1] = PR[GP1:90,1] + 33.066;
   1:  PR[GP1:91,2] = PR[GP1:90,2] + 10.416;
   1:L PR[91] 10mm/sec CNT100;
   1:  PR[GP1:91,1] = PR[GP1:90,1] + 31.921;
   1:  PR[GP1:91,2] = PR[GP1:90,2] + 11.707;
   1:L PR[91] 10mm/sec CNT100;
   1:  PR[GP1:91,1] = PR[GP1:90,1] + 29.327;
   1:  PR[GP1:91,2] = PR[GP1:90,2] + 13.807;
   1:L PR[91] 10mm/sec CNT100;
   1:  PR[GP1:91,1] = PR[GP1:90,1] + 26.380;
   1:  PR[GP1:91,2] = PR[GP1:90,2] + 15.350;
   1:L PR[91] 10mm/sec CNT100;
   1:  PR[GP1:91,1] = PR[GP1:90,1] + 25.459;
   1:  PR[GP1:91,2] = PR[GP1:90,2] + 15.620;
   1:L PR[91] 10mm/sec CNT100;
   1:  PR[GP1:91,1] = PR[GP1:90,1] + 23.944;
   1:  PR[GP1:91,2] = PR[GP1:90,2] + 16.118;
   1:L PR[91] 10mm/sec CNT100;
   1:  PR[GP1:91,1] = PR[GP1:90,1] + 23.209;
   1:  PR[GP1:91,2] = PR[GP1:90,2] + 16.282;
   1:L PR[91] 10mm/sec CNT100;
   1:  PR[GP1:91,1] = PR[GP1:90,1] + 19.871;
   1:  PR[GP1:91,2] = PR[GP1:90,2] + 16.571;
   1:L PR[91] 10mm/sec CNT100;
   1:  PR[GP1:91,1] = PR[GP1:90,1] + 18.583;
   1:  PR[GP1:91,2] = PR[GP1:90,2] + 16.427;
   1:L PR[91] 10mm/sec CNT100;
   1:  PR[GP1:91,1] = PR[GP1:90,1] + 17.903;
   1:  PR[GP1:91,2] = PR[GP1:90,2] + 16.397;
   1:L PR[91] 10mm/sec CNT100;
   1:  PR[GP1:91,1] = PR[GP1:90,1] + 16.577;
   1:  PR[GP1:91,2] = PR[GP1:90,2] + 16.205;
   1:L PR[91] 10mm/sec CNT100;
   1:  PR[GP1:91,1] = PR[GP1:90,1] + 13.412;
   1:  PR[GP1:91,2] = PR[GP1:90,2] + 15.196;
   1:L PR[91] 10mm/sec CNT100;
   1:  PR[GP1:91,1] = PR[GP1:90,1] + 10.491;
   1:  PR[GP1:91,2] = PR[GP1:90,2] + 13.575;
   1:L PR[91] 10mm/sec CNT100;
   1:  PR[GP1:91,1] = PR[GP1:90,1] + 8.553;
   1:  PR[GP1:91,2] = PR[GP1:90,2] + 11.926;
   1:L PR[91] 10mm/sec CNT100;
   1:  PR[GP1:91,1] = PR[GP1:90,1] + 8.129;
   1:  PR[GP1:91,2] = PR[GP1:90,2] + 11.589;
   1:L PR[91] 10mm/sec CNT100;
   1:  PR[GP1:91,1] = PR[GP1:90,1] + 7.971;
   1:  PR[GP1:91,2] = PR[GP1:90,2] + 11.436;
   1:L PR[91] 10mm/sec CNT100;
   1:  PR[GP1:91,1] = PR[GP1:90,1] + 5.896;
   1:  PR[GP1:91,2] = PR[GP1:90,2] + 8.806;
   1:L PR[91] 10mm/sec CNT100;
   1:  PR[GP1:91,1] = PR[GP1:90,1] + 4.365;
   1:  PR[GP1:91,2] = PR[GP1:90,2] + 5.835;
   1:L PR[91] 10mm/sec CNT100;
   1:  PR[GP1:91,1] = PR[GP1:90,1] + 3.428;
   1:  PR[GP1:91,2] = PR[GP1:90,2] + 2.556;
   1:L PR[91] 10mm/sec CNT100;
   1:  PR[GP1:91,1] = PR[GP1:90,1] + 3.273;
   1:  PR[GP1:91,2] = PR[GP1:90,2] + 2.247;
   1:L PR[91] 10mm/sec CNT100;
   1:  PR[GP1:91,1] = PR[GP1:90,1] + 3.106;
   1:  PR[GP1:91,2] = PR[GP1:90,2] + 1.970;
   1:L PR[91] 10mm/sec CNT100;
   1:  PR[GP1:91,1] = PR[GP1:90,1] + 2.821;
   1:  PR[GP1:91,2] = PR[GP1:90,2] + 1.331;
   1:L PR[91] 10mm/sec CNT100;
   1:  PR[GP1:91,1] = PR[GP1:90,1] + 1.698;
   1:  PR[GP1:91,2] = PR[GP1:90,2] + 0.399;
   1:L PR[91] 10mm/sec CNT100;
   1:  PR[GP1:91,1] = PR[GP1:90,1] + 0.370;
   1:  PR[GP1:91,2] = PR[GP1:90,2] + 0.081;
   1:L PR[91] 10mm/sec CNT100;
   1:  PR[GP1:91,1] = PR[GP1:90,1] + -0.233;
   1:L PR[91] 10mm/sec CNT100;
   1:  PR[GP1:91,1] = PR[GP1:90,1] + -0.867;
   1:  PR[GP1:91,2] = PR[GP1:90,2] + 0.236;
   1:L PR[91] 10mm/sec CNT100;
   1:  PR[GP1:91,1] = PR[GP1:90,1] + -1.098;
   1:  PR[GP1:91,2] = PR[GP1:90,2] + 0.267;
   1:L PR[91] 10mm/sec CNT100;
   1:  PR[GP1:91,1] = PR[GP1:90,1] + -1.341;
   1:  PR[GP1:91,2] = PR[GP1:90,2] + 0.332;
   1:L PR[91] 10mm/sec CNT100;
   1:  PR[GP1:91,1] = PR[GP1:90,1] + -1.620;
   1:  PR[GP1:91,2] = PR[GP1:90,2] + 0.457;
   1:L PR[91] 10mm/sec CNT100;
   1:  PR[GP1:91,1] = PR[GP1:90,1] + -2.428;
   1:  PR[GP1:91,2] = PR[GP1:90,2] + 1.122;
   1:L PR[91] 10mm/sec CNT100;
   1:  PR[GP1:91,1] = PR[GP1:90,1] + -2.682;
   1:  PR[GP1:91,2] = PR[GP1:90,2] + 1.395;
   1:L PR[91] 10mm/sec CNT100;
   1:  PR[GP1:91,1] = PR[GP1:90,1] + -3.022;
   1:  PR[GP1:91,2] = PR[GP1:90,2] + 2.163;
   1:L PR[91] 10mm/sec CNT100;
   1:  PR[GP1:91,1] = PR[GP1:90,1] + -3.113;
   1:  PR[GP1:91,2] = PR[GP1:90,2] + 2.168;
   1:L PR[91] 10mm/sec CNT100;
   1:  PR[GP1:91,1] = PR[GP1:90,1] + -3.651;
   1:  PR[GP1:91,2] = PR[GP1:90,2] + 4.205;
   1:L PR[91] 10mm/sec CNT100;
   1:  PR[GP1:91,1] = PR[GP1:90,1] + -3.744;
   1:  PR[GP1:91,2] = PR[GP1:90,2] + 4.627;
   1:L PR[91] 10mm/sec CNT100;
   1:  PR[GP1:91,1] = PR[GP1:90,1] + -4.014;
   1:  PR[GP1:91,2] = PR[GP1:90,2] + 5.559;
   1:L PR[91] 10mm/sec CNT100;
   1:  PR[GP1:91,1] = PR[GP1:90,1] + -4.855;
   1:  PR[GP1:91,2] = PR[GP1:90,2] + 7.425;
   1:L PR[91] 10mm/sec CNT100;
   1:  PR[GP1:91,1] = PR[GP1:90,1] + -5.277;
   1:  PR[GP1:91,2] = PR[GP1:90,2] + 8.208;
   1:L PR[91] 10mm/sec CNT100;
   1:  PR[GP1:91,1] = PR[GP1:90,1] + -6.446;
   1:  PR[GP1:91,2] = PR[GP1:90,2] + 9.963;
   1:L PR[91] 10mm/sec CNT100;
   1:  PR[GP1:91,1] = PR[GP1:90,1] + -6.960;
   1:  PR[GP1:91,2] = PR[GP1:90,2] + 10.566;
   1:L PR[91] 10mm/sec CNT100;
   1:  PR[GP1:91,1] = PR[GP1:90,1] + -8.445;
   1:  PR[GP1:91,2] = PR[GP1:90,2] + 12.151;
   1:L PR[91] 10mm/sec CNT100;
   1:  PR[GP1:91,1] = PR[GP1:90,1] + -10.782;
   1:  PR[GP1:91,2] = PR[GP1:90,2] + 13.939;
   1:L PR[91] 10mm/sec CNT100;
   1:  PR[GP1:91,1] = PR[GP1:90,1] + -12.750;
   1:  PR[GP1:91,2] = PR[GP1:90,2] + 14.986;
   1:L PR[91] 10mm/sec CNT100;
   1:  PR[GP1:91,1] = PR[GP1:90,1] + -13.356;
   1:  PR[GP1:91,2] = PR[GP1:90,2] + 15.272;
   1:L PR[91] 10mm/sec CNT100;
   1:  PR[GP1:91,1] = PR[GP1:90,1] + -15.517;
   1:  PR[GP1:91,2] = PR[GP1:90,2] + 15.997;
   1:L PR[91] 10mm/sec CNT100;
   1:  PR[GP1:91,1] = PR[GP1:90,1] + -16.098;
   1:  PR[GP1:91,2] = PR[GP1:90,2] + 16.133;
   1:L PR[91] 10mm/sec CNT100;
   1:  PR[GP1:91,1] = PR[GP1:90,1] + -18.382;
   1:  PR[GP1:91,2] = PR[GP1:90,2] + 16.500;
   1:L PR[91] 10mm/sec CNT100;
   1:  PR[GP1:91,1] = PR[GP1:90,1] + -20.726;
   1:  PR[GP1:91,2] = PR[GP1:90,2] + 16.487;
   1:L PR[91] 10mm/sec CNT100;
   1:  PR[GP1:91,1] = PR[GP1:90,1] + -21.298;
   1:  PR[GP1:91,2] = PR[GP1:90,2] + 16.496;
   1:L PR[91] 10mm/sec CNT100;
   1:  PR[GP1:91,1] = PR[GP1:90,1] + -23.621;
   1:  PR[GP1:91,2] = PR[GP1:90,2] + 16.097;
   1:L PR[91] 10mm/sec CNT100;
   1:  PR[GP1:91,1] = PR[GP1:90,1] + -24.131;
   1:  PR[GP1:91,2] = PR[GP1:90,2] + 15.996;
   1:L PR[91] 10mm/sec CNT100;
   1:  PR[GP1:91,1] = PR[GP1:90,1] + -26.383;
   1:  PR[GP1:91,2] = PR[GP1:90,2] + 15.212;
   1:L PR[91] 10mm/sec CNT100;
   1:  PR[GP1:91,1] = PR[GP1:90,1] + -26.824;
   1:  PR[GP1:91,2] = PR[GP1:90,2] + 15.023;
   1:L PR[91] 10mm/sec CNT100;
   1:  PR[GP1:91,1] = PR[GP1:90,1] + -28.935;
   1:  PR[GP1:91,2] = PR[GP1:90,2] + 13.870;
   1:L PR[91] 10mm/sec CNT100;
   1:  PR[GP1:91,1] = PR[GP1:90,1] + -29.303;
   1:  PR[GP1:91,2] = PR[GP1:90,2] + 13.608;
   1:L PR[91] 10mm/sec CNT100;
   1:  PR[GP1:91,1] = PR[GP1:90,1] + -31.209;
   1:  PR[GP1:91,2] = PR[GP1:90,2] + 12.115;
   1:L PR[91] 10mm/sec CNT100;
   1:  PR[GP1:91,1] = PR[GP1:90,1] + -33.154;
   1:  PR[GP1:91,2] = PR[GP1:90,2] + 9.991;
   1:L PR[91] 10mm/sec CNT100;
   1:  PR[GP1:91,1] = PR[GP1:90,1] + -34.479;
   1:  PR[GP1:91,2] = PR[GP1:90,2] + 7.952;
   1:L PR[91] 10mm/sec CNT100;
   1:  PR[GP1:91,1] = PR[GP1:90,1] + -34.696;
   1:  PR[GP1:91,2] = PR[GP1:90,2] + 7.582;
   1:L PR[91] 10mm/sec CNT100;
   1:  PR[GP1:91,1] = PR[GP1:90,1] + -35.672;
   1:  PR[GP1:91,2] = PR[GP1:90,2] + 5.348;
   1:L PR[91] 10mm/sec CNT100;
   1:  PR[GP1:91,1] = PR[GP1:90,1] + -35.805;
   1:  PR[GP1:91,2] = PR[GP1:90,2] + 4.945;
   1:L PR[91] 10mm/sec CNT100;
   1:  PR[GP1:91,1] = PR[GP1:90,1] + -36.399;
   1:  PR[GP1:91,2] = PR[GP1:90,2] + 2.589;
   1:L PR[91] 10mm/sec CNT100;
   1:  PR[GP1:91,1] = PR[GP1:90,1] + -36.646;
   1:  PR[GP1:91,2] = PR[GP1:90,2] + -0.278;
   1:L PR[91] 10mm/sec CNT100;
   1:  PR[GP1:91,1] = PR[GP1:90,1] + -36.446;
   1:  PR[GP1:91,2] = PR[GP1:90,2] + -2.707;
   1:L PR[91] 10mm/sec CNT100;
   1:  PR[GP1:91,1] = PR[GP1:90,1] + -36.399;
   1:  PR[GP1:91,2] = PR[GP1:90,2] + -3.140;
   1:L PR[91] 10mm/sec CNT100;
   1:  PR[GP1:91,1] = PR[GP1:90,1] + -35.806;
   1:  PR[GP1:91,2] = PR[GP1:90,2] + -5.489;
   1:L PR[91] 10mm/sec CNT100;
   1:  PR[GP1:91,1] = PR[GP1:90,1] + -35.665;
   1:  PR[GP1:91,2] = PR[GP1:90,2] + -5.918;
   1:L PR[91] 10mm/sec CNT100;
   1:  PR[GP1:91,1] = PR[GP1:90,1] + -34.701;
   1:  PR[GP1:91,2] = PR[GP1:90,2] + -8.125;
   1:L PR[91] 10mm/sec CNT100;
   1:  PR[GP1:91,1] = PR[GP1:90,1] + -34.458;
   1:  PR[GP1:91,2] = PR[GP1:90,2] + -8.539;
   1:L PR[91] 10mm/sec CNT100;
   1:  PR[GP1:91,1] = PR[GP1:90,1] + -33.156;
   1:  PR[GP1:91,2] = PR[GP1:90,2] + -10.540;
   1:L PR[91] 10mm/sec CNT100;
   1:  PR[GP1:91,1] = PR[GP1:90,1] + -31.199;
   1:  PR[GP1:91,2] = PR[GP1:90,2] + -12.676;
   1:L PR[91] 10mm/sec CNT100;
   1:  PR[GP1:91,1] = PR[GP1:90,1] + -29.342;
   1:  PR[GP1:91,2] = PR[GP1:90,2] + -14.131;
   1:L PR[91] 10mm/sec CNT100;
   1:  PR[GP1:91,1] = PR[GP1:90,1] + -28.902;
   1:  PR[GP1:91,2] = PR[GP1:90,2] + -14.442;
   1:L PR[91] 10mm/sec CNT100;
   1:  PR[GP1:91,1] = PR[GP1:90,1] + -26.860;
   1:  PR[GP1:91,2] = PR[GP1:90,2] + -15.557;
   1:L PR[91] 10mm/sec CNT100;
   1:  PR[GP1:91,1] = PR[GP1:90,1] + -26.310;
   1:  PR[GP1:91,2] = PR[GP1:90,2] + -15.791;
   1:L PR[91] 10mm/sec CNT100;
   1:  PR[GP1:91,1] = PR[GP1:90,1] + -24.159;
   1:  PR[GP1:91,2] = PR[GP1:90,2] + -16.540;
   1:L PR[91] 10mm/sec CNT100;
   1:  PR[GP1:91,1] = PR[GP1:90,1] + -22.581;
   1:  PR[GP1:91,2] = PR[GP1:90,2] + -16.804;
   1:  PR[GP1:91,3] = PR[GP1:90,3] + 6.600;
   1:L PR[91] 10mm/sec CNT100;
   1:  PR[GP1:91,1] = PR[GP1:90,1] + -21.203;
   1:  PR[GP1:91,2] = PR[GP1:90,2] + -17.073;
   1:L PR[91] 10mm/sec CNT100;
   1:  PR[GP1:91,1] = PR[GP1:90,1] + -19.633;
   1:  PR[GP1:91,2] = PR[GP1:90,2] + -17.082;
   1:L PR[91] 10mm/sec CNT100;
   1:  PR[GP1:91,1] = PR[GP1:90,1] + -18.058;
   1:  PR[GP1:91,2] = PR[GP1:90,2] + -17.049;
   1:L PR[91] 10mm/sec CNT100;
   1:  PR[GP1:91,1] = PR[GP1:90,1] + -16.627;
   1:  PR[GP1:91,2] = PR[GP1:90,2] + -16.819;
   1:L PR[91] 10mm/sec CNT100;
   1:  PR[GP1:91,1] = PR[GP1:90,1] + -14.900;
   1:  PR[GP1:91,2] = PR[GP1:90,2] + -16.408;
   1:L PR[91] 10mm/sec CNT100;
   1:  PR[GP1:91,1] = PR[GP1:90,1] + -13.653;
   1:  PR[GP1:91,2] = PR[GP1:90,2] + -15.989;
   1:L PR[91] 10mm/sec CNT100;
   1:  PR[GP1:91,1] = PR[GP1:90,1] + -11.859;
   1:  PR[GP1:91,2] = PR[GP1:90,2] + -15.132;
   1:L PR[91] 10mm/sec CNT100;
   1:  PR[GP1:91,1] = PR[GP1:90,1] + -10.818;
   1:  PR[GP1:91,2] = PR[GP1:90,2] + -14.579;
   1:L PR[91] 10mm/sec CNT100;
   1:  PR[GP1:91,1] = PR[GP1:90,1] + -8.234;
   1:  PR[GP1:91,2] = PR[GP1:90,2] + -12.593;
   1:L PR[91] 10mm/sec CNT100;
   1:  PR[GP1:91,1] = PR[GP1:90,1] + -7.515;
   1:  PR[GP1:91,2] = PR[GP1:90,2] + -11.825;
   1:L PR[91] 10mm/sec CNT100;
   1:  PR[GP1:91,1] = PR[GP1:90,1] + -6.063;
   1:  PR[GP1:91,2] = PR[GP1:90,2] + -10.107;
   1:L PR[91] 10mm/sec CNT100;
   1:  PR[GP1:91,1] = PR[GP1:90,1] + -5.533;
   1:  PR[GP1:91,2] = PR[GP1:90,2] + -9.311;
   1:L PR[91] 10mm/sec CNT100;
   1:  PR[GP1:91,1] = PR[GP1:90,1] + -4.418;
   1:  PR[GP1:91,2] = PR[GP1:90,2] + -7.222;
   1:L PR[91] 10mm/sec CNT100;
   1:  PR[GP1:91,1] = PR[GP1:90,1] + -4.048;
   1:  PR[GP1:91,2] = PR[GP1:90,2] + -6.402;
   1:L PR[91] 10mm/sec CNT100;
   1:  PR[GP1:91,1] = PR[GP1:90,1] + -3.149;
   1:  PR[GP1:91,2] = PR[GP1:90,2] + -3.037;
   1:L PR[91] 10mm/sec CNT100;
   1:  PR[GP1:91,1] = PR[GP1:90,1] + -3.006;
   1:  PR[GP1:91,2] = PR[GP1:90,2] + -2.841;
   1:L PR[91] 10mm/sec CNT100;
   1:  PR[GP1:91,1] = PR[GP1:90,1] + -2.754;
   1:  PR[GP1:91,2] = PR[GP1:90,2] + -2.230;
   1:L PR[91] 10mm/sec CNT100;
   1:  PR[GP1:91,1] = PR[GP1:90,1] + -2.624;
   1:  PR[GP1:91,2] = PR[GP1:90,2] + -1.981;
   1:L PR[91] 10mm/sec CNT100;
   1:  PR[GP1:91,1] = PR[GP1:90,1] + -2.404;
   1:  PR[GP1:91,2] = PR[GP1:90,2] + -1.685;
   1:L PR[91] 10mm/sec CNT100;
   1:  PR[GP1:91,1] = PR[GP1:90,1] + -2.028;
   1:  PR[GP1:91,2] = PR[GP1:90,2] + -1.370;
   1:L PR[91] 10mm/sec CNT100;
   1:  PR[GP1:91,1] = PR[GP1:90,1] + -1.921;
   1:  PR[GP1:91,2] = PR[GP1:90,2] + -1.255;
   1:L PR[91] 10mm/sec CNT100;
   1:  PR[GP1:91,1] = PR[GP1:90,1] + -1.712;
   1:  PR[GP1:91,2] = PR[GP1:90,2] + -1.085;
   1:L PR[91] 10mm/sec CNT100;
   1:  PR[GP1:91,1] = PR[GP1:90,1] + -1.397;
   1:  PR[GP1:91,2] = PR[GP1:90,2] + -0.896;
   1:L PR[91] 10mm/sec CNT100;
   1:  PR[GP1:91,1] = PR[GP1:90,1] + -1.090;
   1:  PR[GP1:91,2] = PR[GP1:90,2] + -0.823;
   1:L PR[91] 10mm/sec CNT100;
   1:  PR[GP1:91,1] = PR[GP1:90,1] + -0.937;
   1:  PR[GP1:91,2] = PR[GP1:90,2] + -0.743;
   1:L PR[91] 10mm/sec CNT100;
   1:  PR[GP1:91,1] = PR[GP1:90,1] + -0.555;
   1:  PR[GP1:91,2] = PR[GP1:90,2] + -0.633;
   1:L PR[91] 10mm/sec CNT100;
   1:  PR[GP1:91,1] = PR[GP1:90,1] + 0.097;
   1:  PR[GP1:91,2] = PR[GP1:90,2] + -0.609;
   1:L PR[91] 10mm/sec CNT100;
   1:  PR[GP1:91,1] = PR[GP1:90,1] + 0.838;
   1:  PR[GP1:91,2] = PR[GP1:90,2] + -0.769;
   1:L PR[91] 10mm/sec CNT100;
   1:  PR[GP1:91,1] = PR[GP1:90,1] + 1.525;
   1:  PR[GP1:91,2] = PR[GP1:90,2] + -1.051;
   1:L PR[91] 10mm/sec CNT100;
   1:  PR[GP1:91,1] = PR[GP1:90,1] + 2.185;
   1:  PR[GP1:91,2] = PR[GP1:90,2] + -1.583;
   1:L PR[91] 10mm/sec CNT100;
   1:  PR[GP1:91,1] = PR[GP1:90,1] + 2.553;
   1:  PR[GP1:91,2] = PR[GP1:90,2] + -1.944;
   1:L PR[91] 10mm/sec CNT100;
   1:  PR[GP1:91,1] = PR[GP1:90,1] + 3.082;
   1:  PR[GP1:91,2] = PR[GP1:90,2] + -3.134;
   1:L PR[91] 10mm/sec CNT100;
   1:  PR[GP1:91,1] = PR[GP1:90,1] + 3.767;
   1:  PR[GP1:91,2] = PR[GP1:90,2] + -5.778;
   1:L PR[91] 10mm/sec CNT100;
   1:  PR[GP1:91,1] = PR[GP1:90,1] + 4.204;
   1:  PR[GP1:91,2] = PR[GP1:90,2] + -6.760;
   1:L PR[91] 10mm/sec CNT100;
   1:  PR[GP1:91,1] = PR[GP1:90,1] + 4.850;
   1:  PR[GP1:91,2] = PR[GP1:90,2] + -8.197;
   1:L PR[91] 10mm/sec CNT100;
   1:  PR[GP1:91,1] = PR[GP1:90,1] + 6.326;
   1:  PR[GP1:91,2] = PR[GP1:90,2] + -10.424;
   1:L PR[91] 10mm/sec CNT100;
   1:  PR[GP1:91,1] = PR[GP1:90,1] + 8.119;
   1:  PR[GP1:91,2] = PR[GP1:90,2] + -12.397;
   1:L PR[91] 10mm/sec CNT100;
   1:  PR[GP1:91,1] = PR[GP1:90,1] + 10.182;
   1:  PR[GP1:91,2] = PR[GP1:90,2] + -14.070;
   1:L PR[91] 10mm/sec CNT100;
   1:  PR[GP1:91,1] = PR[GP1:90,1] + 12.482;
   1:  PR[GP1:91,2] = PR[GP1:90,2] + -15.405;
   1:L PR[91] 10mm/sec CNT100;
   1:  PR[GP1:91,1] = PR[GP1:90,1] + 14.967;
   1:  PR[GP1:91,2] = PR[GP1:90,2] + -16.371;
   1:L PR[91] 10mm/sec CNT100;
   1:  PR[GP1:91,1] = PR[GP1:90,1] + 17.497;
   1:  PR[GP1:91,2] = PR[GP1:90,2] + -16.941;
   1:L PR[91] 10mm/sec CNT100;
   1:  PR[GP1:91,1] = PR[GP1:90,1] + 19.904;
   1:  PR[GP1:91,2] = PR[GP1:90,2] + -17.119;
   1:L PR[91] 10mm/sec CNT100;
   1:  PR[GP1:91,1] = PR[GP1:90,1] + 20.243;
   1:  PR[GP1:91,2] = PR[GP1:90,2] + -17.127;
   1:L PR[91] 10mm/sec CNT100;
   1:  PR[GP1:91,1] = PR[GP1:90,1] + 22.689;
   1:  PR[GP1:91,2] = PR[GP1:90,2] + -16.912;
   1:L PR[91] 10mm/sec CNT100;
   1:  PR[GP1:91,1] = PR[GP1:90,1] + 23.204;
   1:  PR[GP1:91,2] = PR[GP1:90,2] + -16.809;
   1:L PR[91] 10mm/sec CNT100;
   1:  PR[GP1:91,1] = PR[GP1:90,1] + 24.937;
   1:  PR[GP1:91,2] = PR[GP1:90,2] + -16.380;
   1:L PR[91] 10mm/sec CNT100;
   1:  PR[GP1:91,1] = PR[GP1:90,1] + 25.573;
   1:  PR[GP1:91,2] = PR[GP1:90,2] + -16.178;
   1:L PR[91] 10mm/sec CNT100;
   1:  PR[GP1:91,1] = PR[GP1:90,1] + 27.731;
   1:  PR[GP1:91,2] = PR[GP1:90,2] + -15.251;
   1:L PR[91] 10mm/sec CNT100;
   1:  PR[GP1:91,1] = PR[GP1:90,1] + 28.409;
   1:  PR[GP1:91,2] = PR[GP1:90,2] + -14.856;
   1:L PR[91] 10mm/sec CNT100;
   1:  PR[GP1:91,1] = PR[GP1:90,1] + 29.656;
   1:  PR[GP1:91,2] = PR[GP1:90,2] + -14.082;
   1:L PR[91] 10mm/sec CNT100;
   1:  PR[GP1:91,1] = PR[GP1:90,1] + 30.356;
   1:  PR[GP1:91,2] = PR[GP1:90,2] + -13.563;
   1:L PR[91] 10mm/sec CNT100;
   1:  PR[GP1:91,1] = PR[GP1:90,1] + 31.356;
   1:  PR[GP1:91,2] = PR[GP1:90,2] + -12.700;
   1:L PR[91] 10mm/sec CNT100;
   1:  PR[GP1:91,1] = PR[GP1:90,1] + 32.048;
   1:  PR[GP1:91,2] = PR[GP1:90,2] + -12.060;
   1:L PR[91] 10mm/sec CNT100;
   1:  PR[GP1:91,1] = PR[GP1:90,1] + 33.492;
   1:  PR[GP1:91,2] = PR[GP1:90,2] + -10.370;
   1:L PR[91] 10mm/sec CNT100;
   1:  PR[GP1:91,1] = PR[GP1:90,1] + 34.057;
   1:  PR[GP1:91,2] = PR[GP1:90,2] + -9.551;
   1:L PR[91] 10mm/sec CNT100;
   1:  PR[GP1:91,1] = PR[GP1:90,1] + 34.667;
   1:  PR[GP1:91,2] = PR[GP1:90,2] + -8.547;
   1:L PR[91] 10mm/sec CNT100;
   1:  PR[GP1:91,1] = PR[GP1:90,1] + 35.159;
   1:  PR[GP1:91,2] = PR[GP1:90,2] + -7.634;
   1:L PR[91] 10mm/sec CNT100;
   1:  PR[GP1:91,1] = PR[GP1:90,1] + 35.988;
   1:  PR[GP1:91,2] = PR[GP1:90,2] + -5.602;
   1:L PR[91] 10mm/sec CNT100;
   1:  PR[GP1:91,1] = PR[GP1:90,1] + 36.278;
   1:  PR[GP1:91,2] = PR[GP1:90,2] + -4.572;
   1:L PR[91] 10mm/sec CNT100;
   1:  PR[GP1:91,1] = PR[GP1:90,1] + 36.530;
   1:  PR[GP1:91,2] = PR[GP1:90,2] + -3.512;
   1:L PR[91] 10mm/sec CNT100;
   1:  PR[GP1:91,1] = PR[GP1:90,1] + 36.707;
   1:  PR[GP1:91,2] = PR[GP1:90,2] + -2.443;
   1:L PR[91] 10mm/sec CNT100;
   1:  PR[GP1:91,1] = PR[GP1:90,1] + 36.769;
   1:  PR[GP1:91,2] = PR[GP1:90,2] + -1.325;
   1:L PR[91] 10mm/sec CNT100;
   1:  PR[GP1:91,1] = PR[GP1:90,1] + 36.871;
   1:  PR[GP1:91,2] = PR[GP1:90,2] + -0.271;
   1:L PR[91] 10mm/sec CNT100;
   1:  PR[GP1:91,1] = PR[GP1:90,1] + 36.528;
   1:  PR[GP1:91,2] = PR[GP1:90,2] + 3.036;
   1:L PR[91] 10mm/sec CNT100;
   1:  PR[GP1:91,1] = PR[GP1:90,1] + 36.106;
   1:  PR[GP1:91,2] = PR[GP1:90,2] + 4.412;
   1:L PR[91] 10mm/sec CNT100;
   1:  PR[GP1:91,1] = PR[GP1:90,1] + 35.770;
   1:  PR[GP1:91,2] = PR[GP1:90,2] + 5.657;
   1:L PR[91] 10mm/sec CNT100;
   1:  PR[GP1:91,1] = PR[GP1:90,1] + 35.564;
   1:  PR[GP1:91,2] = PR[GP1:90,2] + 6.201;
   1:L PR[91] 10mm/sec CNT100;
   1:  PR[GP1:91,1] = PR[GP1:90,1] + 33.973;
   1:  PR[GP1:91,2] = PR[GP1:90,2] + 9.148;
   1:L PR[91] 10mm/sec CNT100;
   1:  PR[GP1:91,1] = PR[GP1:90,1] + 32.965;
   1:  PR[GP1:91,2] = PR[GP1:90,2] + 10.361;
   1:L PR[91] 10mm/sec CNT100;
   1:  PR[GP1:91,1] = PR[GP1:90,1] + 32.614;
   1:  PR[GP1:91,2] = PR[GP1:90,2] + 10.846;
   1:L PR[91] 10mm/sec CNT100;
   1:  PR[GP1:91,1] = PR[GP1:90,1] + 31.856;
   1:  PR[GP1:91,2] = PR[GP1:90,2] + 11.702;
   1:L PR[91] 10mm/sec CNT100;
   1:  PR[GP1:91,1] = PR[GP1:90,1] + 29.261;
   1:  PR[GP1:91,2] = PR[GP1:90,2] + 13.801;
   1:L PR[91] 10mm/sec CNT100;
   1:  PR[GP1:91,1] = PR[GP1:90,1] + 26.314;
   1:  PR[GP1:91,2] = PR[GP1:90,2] + 15.345;
   1:L PR[91] 10mm/sec CNT100;
   1:  PR[GP1:91,1] = PR[GP1:90,1] + 24.267;
   1:  PR[GP1:91,2] = PR[GP1:90,2] + 15.944;
   1:L PR[91] 10mm/sec CNT100;
   1:  PR[GP1:91,1] = PR[GP1:90,1] + 23.490;
   1:  PR[GP1:91,2] = PR[GP1:90,2] + 16.200;
   1:L PR[91] 10mm/sec CNT100;
   1:  PR[GP1:91,1] = PR[GP1:90,1] + 23.145;
   1:  PR[GP1:91,2] = PR[GP1:90,2] + 16.276;
   1:L PR[91] 10mm/sec CNT100;
   1:  PR[GP1:91,1] = PR[GP1:90,1] + 19.803;
   1:  PR[GP1:91,2] = PR[GP1:90,2] + 16.565;
   1:L PR[91] 10mm/sec CNT100;
   1:  PR[GP1:91,1] = PR[GP1:90,1] + 16.974;
   1:  PR[GP1:91,2] = PR[GP1:90,2] + 16.249;
   1:L PR[91] 10mm/sec CNT100;
   1:  PR[GP1:91,1] = PR[GP1:90,1] + 16.801;
   1:  PR[GP1:91,2] = PR[GP1:90,2] + 16.241;
   1:L PR[91] 10mm/sec CNT100;
   1:  PR[GP1:91,1] = PR[GP1:90,1] + 16.512;
   1:  PR[GP1:91,2] = PR[GP1:90,2] + 16.199;
   1:L PR[91] 10mm/sec CNT100;
   1:  PR[GP1:91,1] = PR[GP1:90,1] + 13.329;
   1:  PR[GP1:91,2] = PR[GP1:90,2] + 15.183;
   1:L PR[91] 10mm/sec CNT100;
   1:  PR[GP1:91,1] = PR[GP1:90,1] + 10.373;
   1:  PR[GP1:91,2] = PR[GP1:90,2] + 13.562;
   1:L PR[91] 10mm/sec CNT100;
   1:  PR[GP1:91,1] = PR[GP1:90,1] + 7.800;
   1:  PR[GP1:91,2] = PR[GP1:90,2] + 11.401;
   1:L PR[91] 10mm/sec CNT100;
   1:  PR[GP1:91,1] = PR[GP1:90,1] + 5.699;
   1:  PR[GP1:91,2] = PR[GP1:90,2] + 8.782;
   1:L PR[91] 10mm/sec CNT100;
   1:  PR[GP1:91,1] = PR[GP1:90,1] + 4.116;
   1:  PR[GP1:91,2] = PR[GP1:90,2] + 5.803;
   1:L PR[91] 10mm/sec CNT100;
   1:  PR[GP1:91,1] = PR[GP1:90,1] + 3.143;
   1:  PR[GP1:91,2] = PR[GP1:90,2] + 2.546;
   1:L PR[91] 10mm/sec CNT100;
   1:  PR[GP1:91,1] = PR[GP1:90,1] + 2.595;
   1:  PR[GP1:91,2] = PR[GP1:90,2] + 1.371;
   1:L PR[91] 10mm/sec CNT100;
   1:  PR[GP1:91,1] = PR[GP1:90,1] + 2.311;
   1:  PR[GP1:91,2] = PR[GP1:90,2] + 1.101;
   1:L PR[91] 10mm/sec CNT100;
   1:  PR[GP1:91,1] = PR[GP1:90,1] + 1.548;
   1:  PR[GP1:91,2] = PR[GP1:90,2] + 0.493;
   1:L PR[91] 10mm/sec CNT100;
   1:  PR[GP1:91,1] = PR[GP1:90,1] + 1.020;
   1:  PR[GP1:91,2] = PR[GP1:90,2] + 0.281;
   1:L PR[91] 10mm/sec CNT100;
   1:  PR[GP1:91,1] = PR[GP1:90,1] + 0.227;
   1:  PR[GP1:91,2] = PR[GP1:90,2] + 0.097;
   1:L PR[91] 10mm/sec CNT100;
   1:  PR[GP1:91,1] = PR[GP1:90,1] + -0.121;
   1:  PR[GP1:91,2] = PR[GP1:90,2] + 0.079;
   1:L PR[91] 10mm/sec CNT100;
   1:  PR[GP1:91,1] = PR[GP1:90,1] + -0.724;
   1:  PR[GP1:91,2] = PR[GP1:90,2] + 0.163;
   1:L PR[91] 10mm/sec CNT100;
   1:  PR[GP1:91,1] = PR[GP1:90,1] + -1.140;
   1:  PR[GP1:91,2] = PR[GP1:90,2] + 0.273;
   1:L PR[91] 10mm/sec CNT100;
   1:  PR[GP1:91,1] = PR[GP1:90,1] + -1.595;
   1:  PR[GP1:91,2] = PR[GP1:90,2] + 0.477;
   1:L PR[91] 10mm/sec CNT100;
   1:  PR[GP1:91,1] = PR[GP1:90,1] + -1.963;
   1:  PR[GP1:91,2] = PR[GP1:90,2] + 0.785;
   1:L PR[91] 10mm/sec CNT100;
   1:  PR[GP1:91,1] = PR[GP1:90,1] + -2.160;
   1:  PR[GP1:91,2] = PR[GP1:90,2] + 0.927;
   1:L PR[91] 10mm/sec CNT100;
   1:  PR[GP1:91,1] = PR[GP1:90,1] + -2.422;
   1:  PR[GP1:91,2] = PR[GP1:90,2] + 1.172;
   1:L PR[91] 10mm/sec CNT100;
   1:  PR[GP1:91,1] = PR[GP1:90,1] + -2.634;
   1:  PR[GP1:91,2] = PR[GP1:90,2] + 1.445;
   1:L PR[91] 10mm/sec CNT100;
   1:  PR[GP1:91,1] = PR[GP1:90,1] + -2.875;
   1:  PR[GP1:91,2] = PR[GP1:90,2] + 2.001;
   1:L PR[91] 10mm/sec CNT100;
   1:  PR[GP1:91,1] = PR[GP1:90,1] + -2.961;
   1:  PR[GP1:91,2] = PR[GP1:90,2] + 2.160;
   1:L PR[91] 10mm/sec CNT100;
   1:  PR[GP1:91,1] = PR[GP1:90,1] + -3.091;
   1:  PR[GP1:91,2] = PR[GP1:90,2] + 2.167;
   1:L PR[91] 10mm/sec CNT100;
   1:  PR[GP1:91,1] = PR[GP1:90,1] + -3.437;
   1:  PR[GP1:91,2] = PR[GP1:90,2] + 3.702;
   1:L PR[91] 10mm/sec CNT100;
   1:  PR[GP1:91,1] = PR[GP1:90,1] + -4.043;
   1:  PR[GP1:91,2] = PR[GP1:90,2] + 5.790;
   1:L PR[91] 10mm/sec CNT100;
   1:  PR[GP1:91,1] = PR[GP1:90,1] + -4.520;
   1:  PR[GP1:91,2] = PR[GP1:90,2] + 6.849;
   1:L PR[91] 10mm/sec CNT100;
   1:  PR[GP1:91,1] = PR[GP1:90,1] + -5.461;
   1:  PR[GP1:91,2] = PR[GP1:90,2] + 8.595;
   1:L PR[91] 10mm/sec CNT100;
   1:  PR[GP1:91,1] = PR[GP1:90,1] + -6.180;
   1:  PR[GP1:91,2] = PR[GP1:90,2] + 9.675;
   1:L PR[91] 10mm/sec CNT100;
   1:  PR[GP1:91,1] = PR[GP1:90,1] + -7.330;
   1:  PR[GP1:91,2] = PR[GP1:90,2] + 11.023;
   1:L PR[91] 10mm/sec CNT100;
   1:  PR[GP1:91,1] = PR[GP1:90,1] + -8.309;
   1:  PR[GP1:91,2] = PR[GP1:90,2] + 12.068;
   1:L PR[91] 10mm/sec CNT100;
   1:  PR[GP1:91,1] = PR[GP1:90,1] + -10.806;
   1:  PR[GP1:91,2] = PR[GP1:90,2] + 13.977;
   1:L PR[91] 10mm/sec CNT100;
   1:  PR[GP1:91,1] = PR[GP1:90,1] + -12.180;
   1:  PR[GP1:91,2] = PR[GP1:90,2] + 14.707;
   1:L PR[91] 10mm/sec CNT100;
   1:  PR[GP1:91,1] = PR[GP1:90,1] + -13.544;
   1:  PR[GP1:91,2] = PR[GP1:90,2] + 15.351;
   1:L PR[91] 10mm/sec CNT100;
   1:  PR[GP1:91,1] = PR[GP1:90,1] + -15.121;
   1:  PR[GP1:91,2] = PR[GP1:90,2] + 15.881;
   1:L PR[91] 10mm/sec CNT100;
   1:  PR[GP1:91,1] = PR[GP1:90,1] + -16.437;
   1:  PR[GP1:91,2] = PR[GP1:90,2] + 16.189;
   1:L PR[91] 10mm/sec CNT100;
   1:  PR[GP1:91,1] = PR[GP1:90,1] + -18.162;
   1:  PR[GP1:91,2] = PR[GP1:90,2] + 16.466;
   1:L PR[91] 10mm/sec CNT100;
   1:  PR[GP1:91,1] = PR[GP1:90,1] + -19.941;
   1:  PR[GP1:91,2] = PR[GP1:90,2] + 16.456;
   1:L PR[91] 10mm/sec CNT100;
   1:  PR[GP1:91,1] = PR[GP1:90,1] + -21.239;
   1:  PR[GP1:91,2] = PR[GP1:90,2] + 16.477;
   1:L PR[91] 10mm/sec CNT100;
   1:  PR[GP1:91,1] = PR[GP1:90,1] + -23.044;
   1:  PR[GP1:91,2] = PR[GP1:90,2] + 16.166;
   1:L PR[91] 10mm/sec CNT100;
   1:  PR[GP1:91,1] = PR[GP1:90,1] + -24.206;
   1:  PR[GP1:91,2] = PR[GP1:90,2] + 15.937;
   1:L PR[91] 10mm/sec CNT100;
   1:  PR[GP1:91,1] = PR[GP1:90,1] + -25.993;
   1:  PR[GP1:91,2] = PR[GP1:90,2] + 15.315;
   1:L PR[91] 10mm/sec CNT100;
   1:  PR[GP1:91,1] = PR[GP1:90,1] + -27.002;
   1:  PR[GP1:91,2] = PR[GP1:90,2] + 14.882;
   1:L PR[91] 10mm/sec CNT100;
   1:  PR[GP1:91,1] = PR[GP1:90,1] + -28.702;
   1:  PR[GP1:91,2] = PR[GP1:90,2] + 13.953;
   1:L PR[91] 10mm/sec CNT100;
   1:  PR[GP1:91,1] = PR[GP1:90,1] + -29.548;
   1:  PR[GP1:91,2] = PR[GP1:90,2] + 13.353;
   1:L PR[91] 10mm/sec CNT100;
   1:  PR[GP1:91,1] = PR[GP1:90,1] + -31.099;
   1:  PR[GP1:91,2] = PR[GP1:90,2] + 12.137;
   1:L PR[91] 10mm/sec CNT100;
   1:  PR[GP1:91,1] = PR[GP1:90,1] + -33.129;
   1:  PR[GP1:91,2] = PR[GP1:90,2] + 9.919;
   1:L PR[91] 10mm/sec CNT100;
   1:  PR[GP1:91,1] = PR[GP1:90,1] + -34.216;
   1:  PR[GP1:91,2] = PR[GP1:90,2] + 8.248;
   1:L PR[91] 10mm/sec CNT100;
   1:  PR[GP1:91,1] = PR[GP1:90,1] + -34.715;
   1:  PR[GP1:91,2] = PR[GP1:90,2] + 7.394;
   1:L PR[91] 10mm/sec CNT100;
   1:  PR[GP1:91,1] = PR[GP1:90,1] + -35.518;
   1:  PR[GP1:91,2] = PR[GP1:90,2] + 5.557;
   1:L PR[91] 10mm/sec CNT100;
   1:  PR[GP1:91,1] = PR[GP1:90,1] + -35.824;
   1:  PR[GP1:91,2] = PR[GP1:90,2] + 4.627;
   1:L PR[91] 10mm/sec CNT100;
   1:  PR[GP1:91,1] = PR[GP1:90,1] + -36.313;
   1:  PR[GP1:91,2] = PR[GP1:90,2] + 2.690;
   1:L PR[91] 10mm/sec CNT100;
   1:  PR[GP1:91,1] = PR[GP1:90,1] + -36.480;
   1:  PR[GP1:91,2] = PR[GP1:90,2] + 0.669;
   1:L PR[91] 10mm/sec CNT100;
   1:  PR[GP1:91,1] = PR[GP1:90,1] + -36.582;
   1:  PR[GP1:91,2] = PR[GP1:90,2] + -0.305;
   1:L PR[91] 10mm/sec CNT100;
   1:  PR[GP1:91,1] = PR[GP1:90,1] + -36.418;
   1:  PR[GP1:91,2] = PR[GP1:90,2] + -2.292;
   1:L PR[91] 10mm/sec CNT100;
   1:  PR[GP1:91,1] = PR[GP1:90,1] + -36.311;
   1:  PR[GP1:91,2] = PR[GP1:90,2] + -3.287;
   1:L PR[91] 10mm/sec CNT100;
   1:  PR[GP1:91,1] = PR[GP1:90,1] + -35.827;
   1:  PR[GP1:91,2] = PR[GP1:90,2] + -5.202;
   1:L PR[91] 10mm/sec CNT100;
   1:  PR[GP1:91,1] = PR[GP1:90,1] + -35.503;
   1:  PR[GP1:91,2] = PR[GP1:90,2] + -6.187;
   1:L PR[91] 10mm/sec CNT100;
   1:  PR[GP1:91,1] = PR[GP1:90,1] + -34.725;
   1:  PR[GP1:91,2] = PR[GP1:90,2] + -7.967;
   1:L PR[91] 10mm/sec CNT100;
   1:  PR[GP1:91,1] = PR[GP1:90,1] + -34.168;
   1:  PR[GP1:91,2] = PR[GP1:90,2] + -8.915;
   1:L PR[91] 10mm/sec CNT100;
   1:  PR[GP1:91,1] = PR[GP1:90,1] + -33.133;
   1:  PR[GP1:91,2] = PR[GP1:90,2] + -10.507;
   1:L PR[91] 10mm/sec CNT100;
   1:  PR[GP1:91,1] = PR[GP1:90,1] + -31.078;
   1:  PR[GP1:91,2] = PR[GP1:90,2] + -12.748;
   1:L PR[91] 10mm/sec CNT100;
   1:  PR[GP1:91,1] = PR[GP1:90,1] + -29.630;
   1:  PR[GP1:91,2] = PR[GP1:90,2] + -13.883;
   1:L PR[91] 10mm/sec CNT100;
   1:  PR[GP1:91,1] = PR[GP1:90,1] + -28.630;
   1:  PR[GP1:91,2] = PR[GP1:90,2] + -14.590;
   1:L PR[91] 10mm/sec CNT100;
   1:  PR[GP1:91,1] = PR[GP1:90,1] + -27.079;
   1:  PR[GP1:91,2] = PR[GP1:90,2] + -15.437;
   1:L PR[91] 10mm/sec CNT100;
   1:  PR[GP1:91,1] = PR[GP1:90,1] + -25.835;
   1:  PR[GP1:91,2] = PR[GP1:90,2] + -15.967;
   1:L PR[91] 10mm/sec CNT100;
   1:  PR[GP1:91,1] = PR[GP1:90,1] + -24.257;
   1:  PR[GP1:91,2] = PR[GP1:90,2] + -16.516;
   1:L PR[91] 10mm/sec CNT100;
   1:  PR[GP1:91,1] = PR[GP1:90,1] + -23.279;
   1:  PR[GP1:91,2] = PR[GP1:90,2] + -16.677;
   1:  PR[GP1:91,3] = PR[GP1:90,3] + 7.700;
   1:L PR[91] 10mm/sec CNT100;
   1:  PR[GP1:91,1] = PR[GP1:90,1] + -21.133;
   1:  PR[GP1:91,2] = PR[GP1:90,2] + -17.095;
   1:L PR[91] 10mm/sec CNT100;
   1:  PR[GP1:91,1] = PR[GP1:90,1] + -20.227;
   1:  PR[GP1:91,2] = PR[GP1:90,2] + -17.100;
